	W =  90.000 deg,	P =   0.000 deg,	R =   90.000 deg
};
P[162]{
   GP1:
	UF : 0, UT : 6,		CONFIG : 'N U T, 0, 0, 0',
	X =  224.788  mm,	Y =   -210.243  mm,	Z =   -315.143  mm,
	W =  90.000 deg,	P =   0.000 deg,	R =   90.000 deg
};
P[163]{
   GP1:
	UF : 0, UT : 6,		CONFIG : 'N U T, 0, 0, 0',
	X =  225.758  mm,	Y =   -210.112  mm,	Z =   -326.969  mm,
	W =  90.000 deg,	P =   0.000 deg,	R =   90.000 deg
};
P[164]{
   GP1:
	UF : 0, UT : 6,		CONFIG : 'N U T, 0, 0, 0',
	X =  227.303  mm,	Y =   -209.130  mm,	Z =   -310.855  mm,
	W =  90.000 deg,	P =   0.000 deg,	R =   90.000 deg
};
P[165]{
   GP1:
	UF : 0, UT : 6,		CONFIG : 'N U T, 0, 0, 0',
	X =  228.509  mm,	Y =   -208.538  mm,	Z =   -324.467  mm,
	W =  90.000 deg,	P =   0.000 deg,	R =   90.000 deg
};
P[166]{
   GP1:
	UF : 0, UT : 6,		CONFIG : 'N U T, 0, 0, 0',
	X =  236.027  mm,	Y =   -221.558  mm,	Z =   -327.535  mm,
	W =  90.000 deg,	P =   0.000 deg,	R =   90.000 deg
};
P[167]{
   GP1:
	UF : 0, UT : 6,		CONFIG : 'N U T, 0, 0, 0',
	X =  234.962  mm,	Y =   -222.199  mm,	Z =   -321.974  mm,
	W =  90.000 deg,	P =   0.000 deg,	R =   90.000 deg
};
P[168]{
   GP1:
	UF : 0, UT : 6,		CONFIG : 'N U T, 0, 0, 0',
	X =  234.137  mm,	Y =   -222.880  mm,	Z =   -315.173  mm,
	W =  90.000 deg,	P =   0.000 deg,	R =   90.000 deg
};
P[169]{
   GP1:
	UF : 0, UT : 6,		CONFIG : 'N U T, 0, 0, 0',
	X =  233.285  mm,	Y =   -223.142  mm,	Z =   -324.709  mm,
	W =  90.000 deg,	P =   0.000 deg,	R =   90.000 deg
};
P[170]{
   GP1:
	UF : 0, UT : 6,		CONFIG : 'N U T, 0, 0, 0',
	X =  232.288  mm,	Y =   -223.625  mm,	Z =   -315.398  mm,
	W =  90.000 deg,	P =   0.000 deg,	R =   90.000 deg
};
P[171]{
   GP1:
	UF : 0, UT : 6,		CONFIG : 'N U T, 0, 0, 0',
	X =  231.126  mm,	Y =   -224.281  mm,	Z =   -313.159  mm,
	W =  90.000 deg,	P =   0.000 deg,	R =   90.000 deg
};
P[172]{
   GP1:
	UF : 0, UT : 6,		CONFIG : 'N U T, 0, 0, 0',
	X =  229.645  mm,	Y =   -224.782  mm,	Z =   -313.757  mm,
	W =  90.000 deg,	P =   0.000 deg,	R =   90.000 deg
};
P[173]{
   GP1:
	UF : 0, UT : 6,		CONFIG : 'N U T, 0, 0, 0',
	X =  228.587  mm,	Y =   -225.643  mm,	Z =   -313.551  mm,
	W =  90.000 deg,	P =   0.000 deg,	R =   90.000 deg
};
P[174]{
   GP1:
	UF : 0, UT : 6,		CONFIG : 'N U T, 0, 0, 0',
	X =  228.149  mm,	Y =   -226.124  mm,	Z =   -327.346  mm,
	W =  90.000 deg,	P =   0.000 deg,	R =   90.000 deg
};
P[175]{
   GP1:
	UF : 0, UT : 6,		CONFIG : 'N U T, 0, 0, 0',
	X =  226.254  mm,	Y =   -226.522  mm,	Z =   -322.702  mm,
	W =  90.000 deg,	P =   0.000 deg,	R =   90.000 deg
};
P[176]{
   GP1:
	UF : 0, UT : 6,		CONFIG : 'N U T, 0, 0, 0',
	X =  225.816  mm,	Y =   -227.611  mm,	Z =   -314.588  mm,
	W =  90.000 deg,	P =   0.000 deg,	R =   90.000 deg
};
P[177]{
   GP1:
	UF : 0, UT : 6,		CONFIG : 'N U T, 0, 0, 0',
	X =  224.558  mm,	Y =   -227.894  mm,	Z =   -320.265  mm,
	W =  90.000 deg,	P =   0.000 deg,	R =   90.000 deg
};
P[178]{
   GP1:
	UF : 0, UT : 6,		CONFIG : 'N U T, 0, 0, 0',
	X =  223.276  mm,	Y =   -228.553  mm,	Z =   -326.960  mm,
	W =  90.000 deg,	P =   0.000 deg,	R =   90.000 deg
};
P[179]{
   GP1:
	UF : 0, UT : 6,		CONFIG : 'N U T, 0, 0, 0',
	X =  222.749  mm,	Y =   -229.227  mm,	Z =   -327.686  mm,
	W =  90.000 deg,	P =   0.000 deg,	R =   90.000 deg
};
P[180]{
   GP1:
	UF : 0, UT : 6,		CONFIG : 'N U T, 0, 0, 0',
	X =  221.839  mm,	Y =   -229.266  mm,	Z =   -311.760  mm,
	W =  90.000 deg,	P =   0.000 deg,	R =   90.000 deg
};
P[181]{
   GP1:
	UF : 0, UT : 6,		CONFIG : 'N U T, 0, 0, 0',
	X =  221.094  mm,	Y =   -230.373  mm,	Z =   -313.022  mm,
	W =  90.000 deg,	P =   0.000 deg,	R =   90.000 deg
};
P[182]{
   GP1:
	UF : 0, UT : 6,		CONFIG : 'N U T, 0, 0, 0',
	X =  220.130  mm,	Y =   -230.437  mm,	Z =   -324.917  mm,
	W =  90.000 deg,	P =   0.000 deg,	R =   90.000 deg
};
P[183]{
   GP1:
	UF : 0, UT : 6,		CONFIG : 'N U T, 0, 0, 0',
	X =  219.359  mm,	Y =   -231.525  mm,	Z =   -324.705  mm,
	W =  90.000 deg,	P =   0.000 deg,	R =   90.000 deg
};
P[184]{
   GP1:
	UF : 0, UT : 6,		CONFIG : 'N U T, 0, 0, 0',
	X =  218.328  mm,	Y =   -231.857  mm,	Z =   -320.733  mm,
	W =  90.000 deg,	P =   0.000 deg,	R =   90.000 deg
};
P[185]{
   GP1:
	UF : 0, UT : 6,		CONFIG : 'N U T, 0, 0, 0',
	X =  217.562  mm,	Y =   -231.833  mm,	Z =   -319.447  mm,
	W =  90.000 deg,	P =   0.000 deg,	R =   90.000 deg
};
P[186]{
   GP1:
	UF : 0, UT : 6,		CONFIG : 'N U T, 0, 0, 0',
	X =  216.888  mm,	Y =   -232.430  mm,	Z =   -311.200  mm,
	W =  90.000 deg,	P =   0.000 deg,	R =   90.000 deg
};
P[187]{
   GP1:
	UF : 0, UT : 6,		CONFIG : 'N U T, 0, 0, 0',
	X =  216.001  mm,	Y =   -232.790  mm,	Z =   -327.443  mm,
	W =  90.000 deg,	P =   0.000 deg,	R =   90.000 deg
};
P[188]{
   GP1:
	UF : 0, UT : 6,		CONFIG : 'N U T, 0, 0, 0',
	X =  214.966  mm,	Y =   -233.495  mm,	Z =   -314.364  mm,
	W =  90.000 deg,	P =   0.000 deg,	R =   90.000 deg
};
P[189]{
   GP1:
	UF : 0, UT : 6,		CONFIG : 'N U T, 0, 0, 0',
	X =  213.340  mm,	Y =   -234.714  mm,	Z =   -322.727  mm,
	W =  90.000 deg,	P =   0.000 deg,	R =   90.000 deg
};
P[190]{
   GP1:
	UF : 0, UT : 6,		CONFIG : 'N U T, 0, 0, 0',
	X =  212.316  mm,	Y =   -234.785  mm,	Z =   -314.035  mm,
	W =  90.000 deg,	P =   0.000 deg,	R =   90.000 deg
};
P[191]{
   GP1:
	UF : 0, UT : 6,		CONFIG : 'N U T, 0, 0, 0',
	X =  211.112  mm,	Y =   -235.761  mm,	Z =   -312.348  mm,
	W =  90.000 deg,	P =   0.000 deg,	R =   90.000 deg
};
P[192]{
   GP1:
	UF : 0, UT : 6,		CONFIG : 'N U T, 0, 0, 0',
	X =  209.960  mm,	Y =   -236.382  mm,	Z =   -315.125  mm,
	W =  90.000 deg,	P =   0.000 deg,	R =   90.000 deg
};
P[193]{
   GP1:
	UF : 0, UT : 6,		CONFIG : 'N U T, 0, 0, 0',
	X =  209.037  mm,	Y =   -237.118  mm,	Z =   -320.198  mm,
	W =  90.000 deg,	P =   0.000 deg,	R =   90.000 deg
};
P[194]{
   GP1:
	UF : 0, UT : 6,		CONFIG : 'N U T, 0, 0, 0',
	X =  208.026  mm,	Y =   -237.481  mm,	Z =   -316.356  mm,
	W =  90.000 deg,	P =   0.000 deg,	R =   90.000 deg
};
P[195]{
   GP1:
	UF : 0, UT : 6,		CONFIG : 'N U T, 0, 0, 0',
	X =  207.935  mm,	Y =   -238.178  mm,	Z =   -325.493  mm,
	W =  90.000 deg,	P =   0.000 deg,	R =   90.000 deg
};
P[196]{
   GP1:
	UF : 0, UT : 6,		CONFIG : 'N U T, 0, 0, 0',
	X =  207.107  mm,	Y =   -237.985  mm,	Z =   -319.169  mm,
	W =  90.000 deg,	P =   0.000 deg,	R =   90.000 deg
};
P[197]{
   GP1:
	UF : 0, UT : 6,		CONFIG : 'N U T, 0, 0, 0',
	X =  207.148  mm,	Y =   -238.292  mm,	Z =   -322.311  mm,
	W =  90.000 deg,	P =   0.000 deg,	R =   90.000 deg
};
P[198]{
   GP1:
	UF : 0, UT : 6,		CONFIG : 'N U T, 0, 0, 0',
	X =  207.193  mm,	Y =   -238.442  mm,	Z =   -317.365  mm,
	W =  90.000 deg,	P =   0.000 deg,	R =   90.000 deg
};
P[199]{
   GP1:
	UF : 0, UT : 6,		CONFIG : 'N U T, 0, 0, 0',
	X =  207.015  mm,	Y =   -238.202  mm,	Z =   -313.956  mm,
	W =  90.000 deg,	P =   0.000 deg,	R =   90.000 deg
};
P[200]{
   GP1:
	UF : 0, UT : 6,		CONFIG : 'N U T, 0, 0, 0',
	X =  206.545  mm,	Y =   -238.830  mm,	Z =   -313.041  mm,
	W =  90.000 deg,	P =   0.000 deg,	R =   90.000 deg
};
P[201]{
   GP1:
	UF : 0, UT : 6,		CONFIG : 'N U T, 0, 0, 0',
	X =  206.046  mm,	Y =   -238.312  mm,	Z =   -321.821  mm,
	W =  90.000 deg,	P =   0.000 deg,	R =   90.000 deg
};
P[202]{
   GP1:
	UF : 0, UT : 6,		CONFIG : 'N U T, 0, 0, 0',
	X =  206.072  mm,	Y =   -238.413  mm,	Z =   -313.566  mm,
	W =  90.000 deg,	P =   0.000 deg,	R =   90.000 deg
};
P[203]{
   GP1:
	UF : 0, UT : 6,		CONFIG : 'N U T, 0, 0, 0',
	X =  206.000  mm,	Y =   -238.618  mm,	Z =   -319.197  mm,
	W =  90.000 deg,	P =   0.000 deg,	R =   90.000 deg
};
P[204]{
   GP1:
	UF : 0, UT : 6,		CONFIG : 'N U T, 0, 0, 0',
	X =  205.360  mm,	Y =   -238.553  mm,	Z =   -323.476  mm,
	W =  90.000 deg,	P =   0.000 deg,	R =   90.000 deg
};
P[205]{
   GP1:
	UF : 0, UT : 6,		CONFIG : 'N U T, 0, 0, 0',
	X =  205.394  mm,	Y =   -238.816  mm,	Z =   -314.327  mm,
	W =  90.000 deg,	P =   0.000 deg,	R =   90.000 deg
};
P[206]{
   GP1:
	UF : 0, UT : 6,		CONFIG : 'N U T, 0, 0, 0',
	X =  205.468  mm,	Y =   -239.148  mm,	Z =   -318.562  mm,
	W =  90.000 deg,	P =   0.000 deg,	R =   90.000 deg
};
P[207]{
   GP1:
	UF : 0, UT : 6,		CONFIG : 'N U T, 0, 0, 0',
	X =  205.209  mm,	Y =   -239.739  mm,	Z =   -324.188  mm,
	W =  90.000 deg,	P =   0.000 deg,	R =   90.000 deg
};
P[208]{
   GP1:
	UF : 0, UT : 6,		CONFIG : 'N U T, 0, 0, 0',
	X =  204.658  mm,	Y =   -239.589  mm,	Z =   -316.726  mm,
	W =  90.000 deg,	P =   0.000 deg,	R =   90.000 deg
};
P[209]{
   GP1:
	UF : 0, UT : 6,		CONFIG : 'N U T, 0, 0, 0',
	X =  203.848  mm,	Y =   -239.576  mm,	Z =   -324.082  mm,
	W =  90.000 deg,	P =   0.000 deg,	R =   90.000 deg
};
P[210]{
   GP1:
	UF : 0, UT : 6,		CONFIG : 'N U T, 0, 0, 0',
	X =  203.724  mm,	Y =   -240.092  mm,	Z =   -313.323  mm,
	W =  90.000 deg,	P =   0.000 deg,	R =   90.000 deg
};
P[211]{
   GP1:
	UF : 0, UT : 6,		CONFIG : 'N U T, 0, 0, 0',
	X =  202.753  mm,	Y =   -240.091  mm,	Z =   -323.496  mm,
	W =  90.000 deg,	P =   0.000 deg,	R =   90.000 deg
};
P[212]{
   GP1:
	UF : 0, UT : 6,		CONFIG : 'N U T, 0, 0, 0',
	X =  202.841  mm,	Y =   -240.719  mm,	Z =   -325.615  mm,
	W =  90.000 deg,	P =   0.000 deg,	R =   90.000 deg
};
P[213]{
   GP1:
	UF : 0, UT : 6,		CONFIG : 'N U T, 0, 0, 0',
	X =  202.714  mm,	Y =   -241.173  mm,	Z =   -323.812  mm,
	W =  90.000 deg,	P =   0.000 deg,	R =   90.000 deg
};
P[214]{
   GP1:
	UF : 0, UT : 6,		CONFIG : 'N U T, 0, 0, 0',
	X =  202.146  mm,	Y =   -240.408  mm,	Z =   -321.973  mm,
	W =  90.000 deg,	P =   0.000 deg,	R =   90.000 deg
};
P[215]{
   GP1:
	UF : 0, UT : 6,		CONFIG : 'N U T, 0, 0, 0',
	X =  202.040  mm,	Y =   -241.144  mm,	Z =   -319.450  mm,
	W =  90.000 deg,	P =   0.000 deg,	R =   90.000 deg
};
P[216]{
   GP1:
	UF : 0, UT : 6,		CONFIG : 'N U T, 0, 0, 0',
	X =  201.603  mm,	Y =   -240.788  mm,	Z =   -326.320  mm,
	W =  90.000 deg,	P =   0.000 deg,	R =   90.000 deg
};
P[217]{
   GP1:
	UF : 0, UT : 6,		CONFIG : 'N U T, 0, 0, 0',
	X =  200.943  mm,	Y =   -241.147  mm,	Z =   -325.486  mm,
	W =  90.000 deg,	P =   0.000 deg,	R =   90.000 deg
};
P[218]{
   GP1:
	UF : 0, UT : 6,		CONFIG : 'N U T, 0, 0, 0',
	X =  201.039  mm,	Y =   -241.818  mm,	Z =   -323.445  mm,
	W =  90.000 deg,	P =   0.000 deg,	R =   90.000 deg
};
P[219]{
   GP1:
	UF : 0, UT : 6,		CONFIG : 'N U T, 0, 0, 0',
	X =  200.525  mm,	Y =   -241.662  mm,	Z =   -318.426  mm,
	W =  90.000 deg,	P =   0.000 deg,	R =   90.000 deg
};
P[220]{
   GP1:
	UF : 0, UT : 6,		CONFIG : 'N U T, 0, 0, 0',
	X =  200.346  mm,	Y =   -242.443  mm,	Z =   -322.944  mm,
	W =  90.000 deg,	P =   0.000 deg,	R =   90.000 deg
};
P[221]{
   GP1:
	UF : 0, UT : 6,		CONFIG : 'N U T, 0, 0, 0',
	X =  199.677  mm,	Y =   -242.289  mm,	Z =   -319.034  mm,
	W =  90.000 deg,	P =   0.000 deg,	R =   90.000 deg
};
P[222]{
   GP1:
	UF : 0, UT : 6,		CONFIG : 'N U T, 0, 0, 0',
	X =  198.880  mm,	Y =   -243.196  mm,	Z =   -312.137  mm,
	W =  90.000 deg,	P =   0.000 deg,	R =   90.000 deg
};
P[223]{
   GP1:
	UF : 0, UT : 6,		CONFIG : 'N U T, 0, 0, 0',
	X =  198.372  mm,	Y =   -242.908  mm,	Z =   -319.670  mm,
	W =  90.000 deg,	P =   0.000 deg,	R =   90.000 deg
};
P[224]{
   GP1:
	UF : 0, UT : 6,		CONFIG : 'N U T, 0, 0, 0',
	X =  197.548  mm,	Y =   -243.227  mm,	Z =   -320.526  mm,
	W =  90.000 deg,	P =   0.000 deg,	R =   90.000 deg
};
P[225]{
   GP1:
	UF : 0, UT : 6,		CONFIG : 'N U T, 0, 0, 0',
	X =  197.608  mm,	Y =   -243.970  mm,	Z =   -310.144  mm,
	W =  90.000 deg,	P =   0.000 deg,	R =   90.000 deg
};
P[226]{
   GP1:
	UF : 0, UT : 6,		CONFIG : 'N U T, 0, 0, 0',
	X =  196.892  mm,	Y =   -244.207  mm,	Z =   -322.889  mm,
	W =  90.000 deg,	P =   0.000 deg,	R =   90.000 deg
};
P[227]{
   GP1:
	UF : 0, UT : 6,		CONFIG : 'N U T, 0, 0, 0',
	X =  195.770  mm,	Y =   -244.534  mm,	Z =   -317.358  mm,
	W =  90.000 deg,	P =   0.000 deg,	R =   90.000 deg
};
P[228]{
   GP1:
	UF : 0, UT : 6,		CONFIG : 'N U T, 0, 0, 0',
	X =  195.153  mm,	Y =   -245.287  mm,	Z =   -316.689  mm,
	W =  90.000 deg,	P =   0.000 deg,	R =   90.000 deg
};
P[229]{
   GP1:
	UF : 0, UT : 6,		CONFIG : 'N U T, 0, 0, 0',
	X =  194.505  mm,	Y =   -244.820  mm,	Z =   -323.698  mm,
	W =  90.000 deg,	P =   0.000 deg,	R =   90.000 deg
};
P[230]{
   GP1:
	UF : 0, UT : 6,		CONFIG : 'N U T, 0, 0, 0',
	X =  194.224  mm,	Y =   -245.716  mm,	Z =   -326.476  mm,
	W =  90.000 deg,	P =   0.000 deg,	R =   90.000 deg
};
P[231]{
   GP1:
	UF : 0, UT : 6,		CONFIG : 'N U T, 0, 0, 0',
	X =  193.462  mm,	Y =   -245.718  mm,	Z =   -315.944  mm,
	W =  90.000 deg,	P =   0.000 deg,	R =   90.000 deg
};
P[232]{
   GP1:
	UF : 0, UT : 6,		CONFIG : 'N U T, 0, 0, 0',
	X =  193.608  mm,	Y =   -246.149  mm,	Z =   -317.665  mm,
	W =  90.000 deg,	P =   0.000 deg,	R =   90.000 deg
};
P[233]{
   GP1:
	UF : 0, UT : 6,		CONFIG : 'N U T, 0, 0, 0',
	X =  192.403  mm,	Y =   -246.571  mm,	Z =   -321.320  mm,
	W =  90.000 deg,	P =   0.000 deg,	R =   90.000 deg
};
P[234]{
   GP1:
	UF : 0, UT : 6,		CONFIG : 'N U T, 0, 0, 0',
	X =  191.248  mm,	Y =   -247.020  mm,	Z =   -319.008  mm,
	W =  90.000 deg,	P =   0.000 deg,	R =   90.000 deg
};
P[235]{
   GP1:
	UF : 0, UT : 6,		CONFIG : 'N U T, 0, 0, 0',
	X =  191.043  mm,	Y =   -247.641  mm,	Z =   -317.853  mm,
	W =  90.000 deg,	P =   0.000 deg,	R =   90.000 deg
};
P[236]{
   GP1:
	UF : 0, UT : 6,		CONFIG : 'N U T, 0, 0, 0',
	X =  190.516  mm,	Y =   -247.406  mm,	Z =   -314.457  mm,
	W =  90.000 deg,	P =   0.000 deg,	R =   90.000 deg
};
P[237]{
   GP1:
	UF : 0, UT : 6,		CONFIG : 'N U T, 0, 0, 0',
	X =  189.836  mm,	Y =   -248.145  mm,	Z =   -315.818  mm,
	W =  90.000 deg,	P =   0.000 deg,	R =   90.000 deg
};
P[238]{
   GP1:
	UF : 0, UT : 6,		CONFIG : 'N U T, 0, 0, 0',
	X =  189.085  mm,	Y =   -248.519  mm,	Z =   -310.157  mm,
	W =  90.000 deg,	P =   0.000 deg,	R =   90.000 deg
};
P[239]{
   GP1:
	UF : 0, UT : 6,		CONFIG : 'N U T, 0, 0, 0',
	X =  188.507  mm,	Y =   -248.566  mm,	Z =   -315.070  mm,
	W =  90.000 deg,	P =   0.000 deg,	R =   90.000 deg
};
P[240]{
   GP1:
	UF : 0, UT : 6,		CONFIG : 'N U T, 0, 0, 0',
	X =  187.787  mm,	Y =   -248.752  mm,	Z =   -325.940  mm,
	W =  90.000 deg,	P =   0.000 deg,	R =   90.000 deg
};
P[241]{
   GP1:
	UF : 0, UT : 6,		CONFIG : 'N U T, 0, 0, 0',
	X =  187.122  mm,	Y =   -249.652  mm,	Z =   -310.999  mm,
	W =  90.000 deg,	P =   0.000 deg,	R =   90.000 deg
};
P[242]{
   GP1:
	UF : 0, UT : 6,		CONFIG : 'N U T, 0, 0, 0',
	X =  186.808  mm,	Y =   -250.365  mm,	Z =   -322.828  mm,
	W =  90.000 deg,	P =   0.000 deg,	R =   90.000 deg
};
P[243]{
   GP1:
	UF : 0, UT : 6,		CONFIG : 'N U T, 0, 0, 0',
	X =  186.334  mm,	Y =   -249.614  mm,	Z =   -326.737  mm,
	W =  90.000 deg,	P =   0.000 deg,	R =   90.000 deg
};
P[244]{
   GP1:
	UF : 0, UT : 6,		CONFIG : 'N U T, 0, 0, 0',
	X =  186.496  mm,	Y =   -249.995  mm,	Z =   -310.681  mm,
	W =  90.000 deg,	P =   0.000 deg,	R =   90.000 deg
};
P[245]{
   GP1:
	UF : 0, UT : 6,		CONFIG : 'N U T, 0, 0, 0',
	X =  185.651  mm,	Y =   -250.675  mm,	Z =   -324.252  mm,
	W =  90.000 deg,	P =   0.000 deg,	R =   90.000 deg
};
P[246]{
   GP1:
	UF : 0, UT : 6,		CONFIG : 'N U T, 0, 0, 0',
	X =  185.181  mm,	Y =   -250.524  mm,	Z =   -319.591  mm,
	W =  90.000 deg,	P =   0.000 deg,	R =   90.000 deg
};
P[247]{
   GP1:
	UF : 0, UT : 6,		CONFIG : 'N U T, 0, 0, 0',
	X =  184.766  mm,	Y =   -251.330  mm,	Z =   -314.019  mm,
	W =  90.000 deg,	P =   0.000 deg,	R =   90.000 deg
};
P[248]{
   GP1:
	UF : 0, UT : 6,		CONFIG : 'N U T, 0, 0, 0',
	X =  184.217  mm,	Y =   -251.057  mm,	Z =   -315.680  mm,
	W =  90.000 deg,	P =   0.000 deg,	R =   90.000 deg
};
P[249]{
   GP1:
	UF : 0, UT : 6,		CONFIG : 'N U T, 0, 0, 0',
	X =  183.503  mm,	Y =   -251.481  mm,	Z =   -319.071  mm,
	W =  90.000 deg,	P =   0.000 deg,	R =   90.000 deg
};
P[250]{
   GP1:
	UF : 0, UT : 6,		CONFIG : 'N U T, 0, 0, 0',
	X =  183.596  mm,	Y =   -252.173  mm,	Z =   -323.935  mm,
	W =  90.000 deg,	P =   0.000 deg,	R =   90.000 deg
};
P[251]{
   GP1:
	UF : 0, UT : 6,		CONFIG : 'N U T, 0, 0, 0',
	X =  182.808  mm,	Y =   -251.854  mm,	Z =   -313.115  mm,
	W =  90.000 deg,	P =   0.000 deg,	R =   90.000 deg
};
P[252]{
   GP1:
	UF : 0, UT : 6,		CONFIG : 'N U T, 0, 0, 0',
	X =  182.519  mm,	Y =   -252.698  mm,	Z =   -311.094  mm,
	W =  90.000 deg,	P =   0.000 deg,	R =   90.000 deg
};
P[253]{
   GP1:
	UF : 0, UT : 6,		CONFIG : 'N U T, 0, 0, 0',
	X =  182.133  mm,	Y =   -252.554  mm,	Z =   -312.961  mm,
	W =  90.000 deg,	P =   0.000 deg,	R =   90.000 deg
};
P[254]{
   GP1:
	UF : 0, UT : 6,		CONFIG : 'N U T, 0, 0, 0',
	X =  181.696  mm,	Y =   -252.481  mm,	Z =   -312.907  mm,
	W =  90.000 deg,	P =   0.000 deg,	R =   90.000 deg
};
P[255]{
   GP1:
	UF : 0, UT : 6,		CONFIG : 'N U T, 0, 0, 0',
	X =  181.475  mm,	Y =   -253.156  mm,	Z =   -318.417  mm,
	W =  90.000 deg,	P =   0.000 deg,	R =   90.000 deg
};
P[256]{
   GP1:
	UF : 0, UT : 6,		CONFIG : 'N U T, 0, 0, 0',
	X =  181.098  mm,	Y =   -252.670  mm,	Z =   -325.683  mm,
	W =  90.000 deg,	P =   0.000 deg,	R =   90.000 deg
};
P[257]{
   GP1:
	UF : 0, UT : 6,		CONFIG : 'N U T, 0, 0, 0',
	X =  180.715  mm,	Y =   -253.461  mm,	Z =   -319.202  mm,
	W =  90.000 deg,	P =   0.000 deg,	R =   90.000 deg
};
P[258]{
   GP1:
	UF : 0, UT : 6,		CONFIG : 'N U T, 0, 0, 0',
	X =  180.117  mm,	Y =   -253.445  mm,	Z =   -316.961  mm,
	W =  90.000 deg,	P =   0.000 deg,	R =   90.000 deg
};
P[259]{
   GP1:
	UF : 0, UT : 6,		CONFIG : 'N U T, 0, 0, 0',
	X =  179.724  mm,	Y =   -253.405  mm,	Z =   -327.050  mm,
	W =  90.000 deg,	P =   0.000 deg,	R =   90.000 deg
};
P[260]{
   GP1:
	UF : 0, UT : 6,		CONFIG : 'N U T, 0, 0, 0',
	X =  179.758  mm,	Y =   -254.263  mm,	Z =   -310.411  mm,
	W =  90.000 deg,	P =   0.000 deg,	R =   90.000 deg
};
P[261]{
   GP1:
	UF : 0, UT : 6,		CONFIG : 'N U T, 0, 0, 0',
	X =  179.421  mm,	Y =   -254.004  mm,	Z =   -316.422  mm,
	W =  90.000 deg,	P =   0.000 deg,	R =   90.000 deg
};
P[262]{
   GP1:
	UF : 0, UT : 6,		CONFIG : 'N U T, 0, 0, 0',
	X =  179.168  mm,	Y =   -254.767  mm,	Z =   -323.170  mm,
	W =  90.000 deg,	P =   0.000 deg,	R =   90.000 deg
};
P[263]{
   GP1:
	UF : 0, UT : 6,		CONFIG : 'N U T, 0, 0, 0',
	X =  178.774  mm,	Y =   -254.695  mm,	Z =   -320.156  mm,
	W =  90.000 deg,	P =   0.000 deg,	R =   90.000 deg
};
P[264]{
   GP1:
	UF : 0, UT : 6,		CONFIG : 'N U T, 0, 0, 0',
	X =  178.329  mm,	Y =   -254.157  mm,	Z =   -322.081  mm,
	W =  90.000 deg,	P =   0.000 deg,	R =   90.000 deg
};
P[265]{
   GP1:
	UF : 0, UT : 6,		CONFIG : 'N U T, 0, 0, 0',
	X =  178.522  mm,	Y =   -254.533  mm,	Z =   -316.123  mm,
	W =  90.000 deg,	P =   0.000 deg,	R =   90.000 deg
};
P[266]{
   GP1:
	UF : 0, UT : 6,		CONFIG : 'N U T, 0, 0, 0',
	X =  177.645  mm,	Y =   -254.955  mm,	Z =   -324.671  mm,
	W =  90.000 deg,	P =   0.000 deg,	R =   90.000 deg
};
P[267]{
   GP1:
	UF : 0, UT : 6,		CONFIG : 'N U T, 0, 0, 0',
	X =  177.564  mm,	Y =   -255.635  mm,	Z =   -326.048  mm,
	W =  90.000 deg,	P =   0.000 deg,	R =   90.000 deg
};
P[268]{
   GP1:
	UF : 0, UT : 6,		CONFIG : 'N U T, 0, 0, 0',
	X =  176.916  mm,	Y =   -255.259  mm,	Z =   -314.337  mm,
	W =  90.000 deg,	P =   0.000 deg,	R =   90.000 deg
};
P[269]{
   GP1:
	UF : 0, UT : 6,		CONFIG : 'N U T, 0, 0, 0',
	X =  176.707  mm,	Y =   -256.020  mm,	Z =   -311.027  mm,
	W =  90.000 deg,	P =   0.000 deg,	R =   90.000 deg
};
P[270]{
   GP1:
	UF : 0, UT : 6,		CONFIG : 'N U T, 0, 0, 0',
	X =  176.355  mm,	Y =   -255.557  mm,	Z =   -312.955  mm,
	W =  90.000 deg,	P =   0.000 deg,	R =   90.000 deg
};
P[271]{
   GP1:
	UF : 0, UT : 6,		CONFIG : 'N U T, 0, 0, 0',
	X =  176.055  mm,	Y =   -256.024  mm,	Z =   -309.916  mm,
	W =  90.000 deg,	P =   0.000 deg,	R =   90.000 deg
};
P[272]{
   GP1:
	UF : 0, UT : 6,		CONFIG : 'N U T, 0, 0, 0',
	X =  176.130  mm,	Y =   -256.296  mm,	Z =   -315.346  mm,
	W =  90.000 deg,	P =   0.000 deg,	R =   90.000 deg
};
P[273]{
   GP1:
	UF : 0, UT : 6,		CONFIG : 'N U T, 0, 0, 0',
	X =  175.786  mm,	Y =   -255.774  mm,	Z =   -322.730  mm,
	W =  90.000 deg,	P =   0.000 deg,	R =   90.000 deg
};
P[274]{
   GP1:
	UF : 0, UT : 6,		CONFIG : 'N U T, 0, 0, 0',
	X =  175.133  mm,	Y =   -256.020  mm,	Z =   -323.009  mm,
	W =  90.000 deg,	P =   0.000 deg,	R =   90.000 deg
};
P[275]{
   GP1:
	UF : 0, UT : 6,		CONFIG : 'N U T, 0, 0, 0',
	X =  175.034  mm,	Y =   -256.520  mm,	Z =   -318.149  mm,
	W =  90.000 deg,	P =   0.000 deg,	R =   90.000 deg
};
P[276]{
   GP1:
	UF : 0, UT : 6,		CONFIG : 'N U T, 0, 0, 0',
	X =  174.768  mm,	Y =   -256.256  mm,	Z =   -327.394  mm,
	W =  90.000 deg,	P =   0.000 deg,	R =   90.000 deg
};
P[277]{
   GP1:
	UF : 0, UT : 6,		CONFIG : 'N U T, 0, 0, 0',
	X =  175.139  mm,	Y =   -257.050  mm,	Z =   -326.450  mm,
	W =  90.000 deg,	P =   0.000 deg,	R =   90.000 deg
};
P[278]{
   GP1:
	UF : 0, UT : 6,		CONFIG : 'N U T, 0, 0, 0',
	X =  174.185  mm,	Y =   -257.011  mm,	Z =   -318.021  mm,
	W =  90.000 deg,	P =   0.000 deg,	R =   90.000 deg
};
P[279]{
   GP1:
	UF : 0, UT : 6,		CONFIG : 'N U T, 0, 0, 0',
	X =  174.073  mm,	Y =   -256.837  mm,	Z =   -310.875  mm,
	W =  90.000 deg,	P =   0.000 deg,	R =   90.000 deg
};
P[280]{
   GP1:
	UF : 0, UT : 6,		CONFIG : 'N U T, 0, 0, 0',
	X =  173.977  mm,	Y =   -256.815  mm,	Z =   -323.368  mm,
	W =  90.000 deg,	P =   0.000 deg,	R =   90.000 deg
};
P[281]{
   GP1:
	UF : 0, UT : 6,		CONFIG : 'N U T, 0, 0, 0',
	X =  174.328  mm,	Y =   -257.478  mm,	Z =   -322.177  mm,
	W =  90.000 deg,	P =   0.000 deg,	R =   90.000 deg
};
P[282]{
   GP1:
	UF : 0, UT : 6,		CONFIG : 'N U T, 0, 0, 0',
	X =  173.792  mm,	Y =   -256.836  mm,	Z =   -326.792  mm,
	W =  90.000 deg,	P =   0.000 deg,	R =   90.000 deg
};
P[283]{
   GP1:
	UF : 0, UT : 6,		CONFIG : 'N U T, 0, 0, 0',
	X =  174.088  mm,	Y =   -257.395  mm,	Z =   -320.324  mm,
	W =  90.000 deg,	P =   0.000 deg,	R =   90.000 deg
};
P[284]{
   GP1:
	UF : 0, UT : 6,		CONFIG : 'N U T, 0, 0, 0',
	X =  173.281  mm,	Y =   -257.367  mm,	Z =   -315.190  mm,
	W =  90.000 deg,	P =   0.000 deg,	R =   90.000 deg
};
P[285]{
   GP1:
	UF : 0, UT : 6,		CONFIG : 'N U T, 0, 0, 0',
	X =  173.246  mm,	Y =   -257.556  mm,	Z =   -317.174  mm,
	W =  90.000 deg,	P =   0.000 deg,	R =   90.000 deg
};
P[286]{
   GP1:
	UF : 0, UT : 6,		CONFIG : 'N U T, 0, 0, 0',
	X =  173.451  mm,	Y =   -258.059  mm,	Z =   -323.350  mm,
	W =  90.000 deg,	P =   0.000 deg,	R =   90.000 deg
};
P[287]{
   GP1:
	UF : 0, UT : 6,		CONFIG : 'N U T, 0, 0, 0',
	X =  172.991  mm,	Y =   -257.452  mm,	Z =   -311.441  mm,
	W =  90.000 deg,	P =   0.000 deg,	R =   90.000 deg
};
P[288]{
   GP1:
	UF : 0, UT : 6,		CONFIG : 'N U T, 0, 0, 0',
	X =  172.967  mm,	Y =   -257.956  mm,	Z =   -327.172  mm,
	W =  90.000 deg,	P =   0.000 deg,	R =   90.000 deg
};
P[289]{
   GP1:
	UF : 0, UT : 6,		CONFIG : 'N U T, 0, 0, 0',
	X =  172.399  mm,	Y =   -258.123  mm,	Z =   -325.331  mm,
	W =  90.000 deg,	P =   0.000 deg,	R =   90.000 deg
};
P[290]{
   GP1:
	UF : 0, UT : 6,		CONFIG : 'N U T, 0, 0, 0',
	X =  172.171  mm,	Y =   -258.662  mm,	Z =   -320.276  mm,
	W =  90.000 deg,	P =   0.000 deg,	R =   90.000 deg
};
P[291]{
   GP1:
	UF : 0, UT : 6,		CONFIG : 'N U T, 0, 0, 0',
	X =  171.769  mm,	Y =   -258.821  mm,	Z =   -313.988  mm,
	W =  90.000 deg,	P =   0.000 deg,	R =   90.000 deg
};
P[292]{
   GP1:
	UF : 0, UT : 6,		CONFIG : 'N U T, 0, 0, 0',
	X =  171.718  mm,	Y =   -258.746  mm,	Z =   -323.267  mm,
	W =  90.000 deg,	P =   0.000 deg,	R =   90.000 deg
};
P[293]{
   GP1:
	UF : 0, UT : 6,		CONFIG : 'N U T, 0, 0, 0',
	X =  171.315  mm,	Y =   -258.833  mm,	Z =   -316.420  mm,
	W =  90.000 deg,	P =   0.000 deg,	R =   90.000 deg
};
P[294]{
   GP1:
	UF : 0, UT : 6,		CONFIG : 'N U T, 0, 0, 0',
	X =  171.438  mm,	Y =   -259.276  mm,	Z =   -321.449  mm,
	W =  90.000 deg,	P =   0.000 deg,	R =   90.000 deg
};
P[295]{
   GP1:
	UF : 0, UT : 6,		CONFIG : 'N U T, 0, 0, 0',
	X =  170.919  mm,	Y =   -259.359  mm,	Z =   -310.652  mm,
	W =  90.000 deg,	P =   0.000 deg,	R =   90.000 deg
};
P[296]{
   GP1:
	UF : 0, UT : 6,		CONFIG : 'N U T, 0, 0, 0',
	X =  170.435  mm,	Y =   -258.753  mm,	Z =   -323.064  mm,
	W =  90.000 deg,	P =   0.000 deg,	R =   90.000 deg
};
P[297]{
   GP1:
	UF : 0, UT : 6,		CONFIG : 'N U T, 0, 0, 0',
	X =  170.812  mm,	Y =   -259.537  mm,	Z =   -326.812  mm,
	W =  90.000 deg,	P =   0.000 deg,	R =   90.000 deg
};
P[298]{
   GP1:
	UF : 0, UT : 6,		CONFIG : 'N U T, 0, 0, 0',
	X =  170.323  mm,	Y =   -259.748  mm,	Z =   -322.919  mm,
	W =  90.000 deg,	P =   0.000 deg,	R =   90.000 deg
};
P[299]{
   GP1:
	UF : 0, UT : 6,		CONFIG : 'N U T, 0, 0, 0',
	X =  169.161  mm,	Y =   -260.175  mm,	Z =   -326.899  mm,
	W =  90.000 deg,	P =   0.000 deg,	R =   90.000 deg
};
P[300]{
   GP1:
	UF : 0, UT : 6,		CONFIG : 'N U T, 0, 0, 0',
	X =  168.079  mm,	Y =   -260.866  mm,	Z =   -320.051  mm,
	W =  90.000 deg,	P =   0.000 deg,	R =   90.000 deg
};
P[301]{
   GP1:
	UF : 0, UT : 6,		CONFIG : 'N U T, 0, 0, 0',
	X =  167.000  mm,	Y =   -261.260  mm,	Z =   -310.192  mm,
	W =  90.000 deg,	P =   0.000 deg,	R =   90.000 deg
};
P[302]{
   GP1:
	UF : 0, UT : 6,		CONFIG : 'N U T, 0, 0, 0',
	X =  165.759  mm,	Y =   -261.835  mm,	Z =   -322.908  mm,
	W =  90.000 deg,	P =   0.000 deg,	R =   90.000 deg
};
P[303]{
   GP1:
	UF : 0, UT : 6,		CONFIG : 'N U T, 0, 0, 0',
	X =  164.606  mm,	Y =   -262.570  mm,	Z =   -315.081  mm,
	W =  90.000 deg,	P =   0.000 deg,	R =   90.000 deg
};
P[304]{
   GP1:
	UF : 0, UT : 6,		CONFIG : 'N U T, 0, 0, 0',
	X =  163.888  mm,	Y =   -263.372  mm,	Z =   -314.268  mm,
	W =  90.000 deg,	P =   0.000 deg,	R =   90.000 deg
};
P[305]{
   GP1:
	UF : 0, UT : 6,		CONFIG : 'N U T, 0, 0, 0',
	X =  163.182  mm,	Y =   -263.663  mm,	Z =   -322.510  mm,
	W =  90.000 deg,	P =   0.000 deg,	R =   90.000 deg
};
P[306]{
   GP1:
	UF : 0, UT : 6,		CONFIG : 'N U T, 0, 0, 0',
	X =  162.268  mm,	Y =   -264.286  mm,	Z =   -315.824  mm,
	W =  90.000 deg,	P =   0.000 deg,	R =   90.000 deg
};
P[307]{
   GP1:
	UF : 0, UT : 6,		CONFIG : 'N U T, 0, 0, 0',
	X =  161.046  mm,	Y =   -264.171  mm,	Z =   -324.463  mm,
	W =  90.000 deg,	P =   0.000 deg,	R =   90.000 deg
};
P[308]{
   GP1:
	UF : 0, UT : 6,		CONFIG : 'N U T, 0, 0, 0',
	X =  160.503  mm,	Y =   -264.987  mm,	Z =   -310.228  mm,
	W =  90.000 deg,	P =   0.000 deg,	R =   90.000 deg
};
P[309]{
   GP1:
	UF : 0, UT : 6,		CONFIG : 'N U T, 0, 0, 0',
	X =  159.727  mm,	Y =   -265.455  mm,	Z =   -311.043  mm,
	W =  90.000 deg,	P =   0.000 deg,	R =   90.000 deg
};
P[310]{
   GP1:
	UF : 0, UT : 6,		CONFIG : 'N U T, 0, 0, 0',
	X =  158.548  mm,	Y =   -265.744  mm,	Z =   -324.807  mm,
	W =  90.000 deg,	P =   0.000 deg,	R =   90.000 deg
};
P[311]{
   GP1:
	UF : 0, UT : 6,		CONFIG : 'N U T, 0, 0, 0',
	X =  157.941  mm,	Y =   -266.872  mm,	Z =   -309.962  mm,
	W =  90.000 deg,	P =   0.000 deg,	R =   90.000 deg
};
P[312]{
   GP1:
	UF : 0, UT : 6,		CONFIG : 'N U T, 0, 0, 0',
	X =  155.789  mm,	Y =   -267.639  mm,	Z =   -316.630  mm,
	W =  90.000 deg,	P =   0.000 deg,	R =   90.000 deg
};
P[313]{
   GP1:
	UF : 0, UT : 6,		CONFIG : 'N U T, 0, 0, 0',
	X =  155.104  mm,	Y =   -268.015  mm,	Z =   -318.141  mm,
	W =  90.000 deg,	P =   0.000 deg,	R =   90.000 deg
};
P[314]{
   GP1:
	UF : 0, UT : 6,		CONFIG : 'N U T, 0, 0, 0',
	X =  154.627  mm,	Y =   -268.796  mm,	Z =   -316.149  mm,
	W =  90.000 deg,	P =   0.000 deg,	R =   90.000 deg
};
P[315]{
   GP1:
	UF : 0, UT : 6,		CONFIG : 'N U T, 0, 0, 0',
	X =  152.644  mm,	Y =   -269.405  mm,	Z =   -325.490  mm,
	W =  90.000 deg,	P =   0.000 deg,	R =   90.000 deg
};
P[316]{
   GP1:
	UF : 0, UT : 6,		CONFIG : 'N U T, 0, 0, 0',
	X =  151.708  mm,	Y =   -270.168  mm,	Z =   -316.163  mm,
	W =  90.000 deg,	P =   0.000 deg,	R =   90.000 deg
};
P[317]{
   GP1:
	UF : 0, UT : 6,		CONFIG : 'N U T, 0, 0, 0',
	X =  151.058  mm,	Y =   -270.792  mm,	Z =   -313.563  mm,
	W =  90.000 deg,	P =   0.000 deg,	R =   90.000 deg
};
P[318]{
   GP1:
	UF : 0, UT : 6,		CONFIG : 'N U T, 0, 0, 0',
	X =  150.279  mm,	Y =   -270.993  mm,	Z =   -316.136  mm,
	W =  90.000 deg,	P =   0.000 deg,	R =   90.000 deg
};
P[319]{
   GP1:
	UF : 0, UT : 6,		CONFIG : 'N U T, 0, 0, 0',
	X =  148.923  mm,	Y =   -271.261  mm,	Z =   -321.051  mm,
	W =  90.000 deg,	P =   0.000 deg,	R =   90.000 deg
};
P[320]{
   GP1:
	UF : 0, UT : 6,		CONFIG : 'N U T, 0, 0, 0',
	X =  148.393  mm,	Y =   -272.295  mm,	Z =   -315.157  mm,
	W =  90.000 deg,	P =   0.000 deg,	R =   90.000 deg
};
P[321]{
   GP1:
	UF : 0, UT : 6,		CONFIG : 'N U T, 0, 0, 0',
	X =  147.670  mm,	Y =   -272.189  mm,	Z =   -320.863  mm,
	W =  90.000 deg,	P =   0.000 deg,	R =   90.000 deg
};
P[322]{
   GP1:
	UF : 0, UT : 6,		CONFIG : 'N U T, 0, 0, 0',
	X =  146.965  mm,	Y =   -273.156  mm,	Z =   -314.071  mm,
	W =  90.000 deg,	P =   0.000 deg,	R =   90.000 deg
};
P[323]{
   GP1:
	UF : 0, UT : 6,		CONFIG : 'N U T, 0, 0, 0',
	X =  145.739  mm,	Y =   -273.756  mm,	Z =   -324.061  mm,
	W =  90.000 deg,	P =   0.000 deg,	R =   90.000 deg
};
P[324]{
   GP1:
	UF : 0, UT : 6,		CONFIG : 'N U T, 0, 0, 0',
	X =  144.779  mm,	Y =   -273.933  mm,	Z =   -324.540  mm,
	W =  90.000 deg,	P =   0.000 deg,	R =   90.000 deg
};
P[325]{
   GP1:
	UF : 0, UT : 6,		CONFIG : 'N U T, 0, 0, 0',
	X =  143.574  mm,	Y =   -274.352  mm,	Z =   -322.371  mm,
	W =  90.000 deg,	P =   0.000 deg,	R =   90.000 deg
};
P[326]{
   GP1:
	UF : 0, UT : 6,		CONFIG : 'N U T, 0, 0, 0',
	X =  143.172  mm,	Y =   -275.465  mm,	Z =   -322.656  mm,
	W =  90.000 deg,	P =   0.000 deg,	R =   90.000 deg
};
P[327]{
   GP1:
	UF : 0, UT : 6,		CONFIG : 'N U T, 0, 0, 0',
	X =  142.457  mm,	Y =   -275.162  mm,	Z =   -314.680  mm,
	W =  90.000 deg,	P =   0.000 deg,	R =   90.000 deg
};
P[328]{
   GP1:
	UF : 0, UT : 6,		CONFIG : 'N U T, 0, 0, 0',
	X =  141.235  mm,	Y =   -276.007  mm,	Z =   -320.583  mm,
	W =  90.000 deg,	P =   0.000 deg,	R =   90.000 deg
};
P[329]{
   GP1:
	UF : 0, UT : 6,		CONFIG : 'N U T, 0, 0, 0',
	X =  139.778  mm,	Y =   -276.839  mm,	Z =   -323.425  mm,
	W =  90.000 deg,	P =   0.000 deg,	R =   90.000 deg
};
P[330]{
   GP1:
	UF : 0, UT : 6,		CONFIG : 'N U T, 0, 0, 0',
	X =  139.030  mm,	Y =   -277.352  mm,	Z =   -312.989  mm,
	W =  90.000 deg,	P =   0.000 deg,	R =   90.000 deg
};
P[331]{
   GP1:
	UF : 0, UT : 6,		CONFIG : 'N U T, 0, 0, 0',
	X =  137.952  mm,	Y =   -277.643  mm,	Z =   -321.278  mm,
	W =  90.000 deg,	P =   0.000 deg,	R =   90.000 deg
};
P[332]{
   GP1:
	UF : 0, UT : 6,		CONFIG : 'N U T, 0, 0, 0',
	X =  136.965  mm,	Y =   -278.708  mm,	Z =   -317.629  mm,
	W =  90.000 deg,	P =   0.000 deg,	R =   90.000 deg
};
P[333]{
   GP1:
	UF : 0, UT : 6,		CONFIG : 'N U T, 0, 0, 0',
	X =  135.994  mm,	Y =   -279.139  mm,	Z =   -309.930  mm,
	W =  90.000 deg,	P =   0.000 deg,	R =   90.000 deg
};
P[334]{
   GP1:
	UF : 0, UT : 6,		CONFIG : 'N U T, 0, 0, 0',
	X =  135.263  mm,	Y =   -279.963  mm,	Z =   -309.813  mm,
	W =  90.000 deg,	P =   0.000 deg,	R =   90.000 deg
};
P[335]{
   GP1:
	UF : 0, UT : 6,		CONFIG : 'N U T, 0, 0, 0',
	X =  134.116  mm,	Y =   -280.032  mm,	Z =   -326.781  mm,
	W =  90.000 deg,	P =   0.000 deg,	R =   90.000 deg
};
P[336]{
   GP1:
	UF : 0, UT : 6,		CONFIG : 'N U T, 0, 0, 0',
	X =  133.461  mm,	Y =   -280.388  mm,	Z =   -319.964  mm,
	W =  90.000 deg,	P =   0.000 deg,	R =   90.000 deg
};
P[337]{
   GP1:
	UF : 0, UT : 6,		CONFIG : 'N U T, 0, 0, 0',
	X =  132.576  mm,	Y =   -281.195  mm,	Z =   -315.012  mm,
	W =  90.000 deg,	P =   0.000 deg,	R =   90.000 deg
};
P[338]{
   GP1:
	UF : 0, UT : 6,		CONFIG : 'N U T, 0, 0, 0',
	X =  131.769  mm,	Y =   -281.560  mm,	Z =   -312.044  mm,
	W =  90.000 deg,	P =   0.000 deg,	R =   90.000 deg
};
P[339]{
   GP1:
	UF : 0, UT : 6,		CONFIG : 'N U T, 0, 0, 0',
	X =  131.139  mm,	Y =   -282.490  mm,	Z =   -324.044  mm,
	W =  90.000 deg,	P =   0.000 deg,	R =   90.000 deg
};
P[340]{
   GP1:
	UF : 0, UT : 6,		CONFIG : 'N U T, 0, 0, 0',
	X =  130.072  mm,	Y =   -282.234  mm,	Z =   -310.531  mm,
	W =  90.000 deg,	P =   0.000 deg,	R =   90.000 deg
};
P[341]{
   GP1:
	UF : 0, UT : 6,		CONFIG : 'N U T, 0, 0, 0',
	X =  129.157  mm,	Y =   -282.609  mm,	Z =   -314.274  mm,
	W =  90.000 deg,	P =   0.000 deg,	R =   90.000 deg
};
P[342]{
   GP1:
	UF : 0, UT : 6,		CONFIG : 'N U T, 0, 0, 0',
	X =  128.370  mm,	Y =   -283.586  mm,	Z =   -312.020  mm,
	W =  90.000 deg,	P =   0.000 deg,	R =   90.000 deg
};
P[343]{
   GP1:
	UF : 0, UT : 6,		CONFIG : 'N U T, 0, 0, 0',
	X =  127.589  mm,	Y =   -284.250  mm,	Z =   -319.858  mm,
	W =  90.000 deg,	P =   0.000 deg,	R =   90.000 deg
};
P[344]{
   GP1:
	UF : 0, UT : 6,		CONFIG : 'N U T, 0, 0, 0',
	X =  126.152  mm,	Y =   -284.494  mm,	Z =   -310.955  mm,
	W =  90.000 deg,	P =   0.000 deg,	R =   90.000 deg
};
P[345]{
   GP1:
	UF : 0, UT : 6,		CONFIG : 'N U T, 0, 0, 0',
	X =  125.723  mm,	Y =   -285.474  mm,	Z =   -309.903  mm,
	W =  90.000 deg,	P =   0.000 deg,	R =   90.000 deg
};
P[346]{
   GP1:
	UF : 0, UT : 6,		CONFIG : 'N U T, 0, 0, 0',
	X =  125.068  mm,	Y =   -285.757  mm,	Z =   -315.898  mm,
	W =  90.000 deg,	P =   0.000 deg,	R =   90.000 deg
};
P[347]{
   GP1:
	UF : 0, UT : 6,		CONFIG : 'N U T, 0, 0, 0',
	X =  125.092  mm,	Y =   -285.932  mm,	Z =   -327.312  mm,
	W =  90.000 deg,	P =   0.000 deg,	R =   90.000 deg
};
P[348]{
   GP1:
	UF : 0, UT : 6,		CONFIG : 'N U T, 0, 0, 0',
	X =  124.931  mm,	Y =   -285.680  mm,	Z =   -320.686  mm,
	W =  90.000 deg,	P =   0.000 deg,	R =   90.000 deg
};
P[349]{
   GP1:
	UF : 0, UT : 6,		CONFIG : 'N U T, 0, 0, 0',
	X =  124.761  mm,	Y =   -285.441  mm,	Z =   -325.611  mm,
	W =  90.000 deg,	P =   0.000 deg,	R =   90.000 deg
};
P[350]{
   GP1:
	UF : 0, UT : 6,		CONFIG : 'N U T, 0, 0, 0',
	X =  124.699  mm,	Y =   -286.144  mm,	Z =   -323.532  mm,
	W =  90.000 deg,	P =   0.000 deg,	R =   90.000 deg
};
P[351]{
   GP1:
	UF : 0, UT : 6,		CONFIG : 'N U T, 0, 0, 0',
	X =  124.243  mm,	Y =   -285.790  mm,	Z =   -322.352  mm,
	W =  90.000 deg,	P =   0.000 deg,	R =   90.000 deg
};
P[352]{
   GP1:
	UF : 0, UT : 6,		CONFIG : 'N U T, 0, 0, 0',
	X =  124.070  mm,	Y =   -285.713  mm,	Z =   -312.258  mm,
	W =  90.000 deg,	P =   0.000 deg,	R =   90.000 deg
};
P[353]{
   GP1:
	UF : 0, UT : 6,		CONFIG : 'N U T, 0, 0, 0',
	X =  124.173  mm,	Y =   -286.448  mm,	Z =   -324.680  mm,
	W =  90.000 deg,	P =   0.000 deg,	R =   90.000 deg
};
P[354]{
   GP1:
	UF : 0, UT : 6,		CONFIG : 'N U T, 0, 0, 0',
	X =  123.770  mm,	Y =   -285.969  mm,	Z =   -317.711  mm,
	W =  90.000 deg,	P =   0.000 deg,	R =   90.000 deg
};
P[355]{
   GP1:
	UF : 0, UT : 6,		CONFIG : 'N U T, 0, 0, 0',
	X =  123.819  mm,	Y =   -286.246  mm,	Z =   -313.172  mm,
	W =  90.000 deg,	P =   0.000 deg,	R =   90.000 deg
};
P[356]{
   GP1:
	UF : 0, UT : 6,		CONFIG : 'N U T, 0, 0, 0',
	X =  123.124  mm,	Y =   -286.169  mm,	Z =   -321.304  mm,
	W =  90.000 deg,	P =   0.000 deg,	R =   90.000 deg
};
P[357]{
   GP1:
	UF : 0, UT : 6,		CONFIG : 'N U T, 0, 0, 0',
	X =  123.054  mm,	Y =   -286.394  mm,	Z =   -319.367  mm,
	W =  90.000 deg,	P =   0.000 deg,	R =   90.000 deg
};
P[358]{
   GP1:
	UF : 0, UT : 6,		CONFIG : 'N U T, 0, 0, 0',
	X =  123.154  mm,	Y =   -286.634  mm,	Z =   -314.348  mm,
	W =  90.000 deg,	P =   0.000 deg,	R =   90.000 deg
};
P[359]{
   GP1:
	UF : 0, UT : 6,		CONFIG : 'N U T, 0, 0, 0',
	X =  123.216  mm,	Y =   -286.990  mm,	Z =   -321.318  mm,
	W =  90.000 deg,	P =   0.000 deg,	R =   90.000 deg
};
P[360]{
   GP1:
	UF : 0, UT : 6,		CONFIG : 'N U T, 0, 0, 0',
	X =  122.488  mm,	Y =   -286.848  mm,	Z =   -318.482  mm,
	W =  90.000 deg,	P =   0.000 deg,	R =   90.000 deg
};
P[361]{
   GP1:
	UF : 0, UT : 6,		CONFIG : 'N U T, 0, 0, 0',
	X =  122.626  mm,	Y =   -287.393  mm,	Z =   -327.120  mm,
	W =  90.000 deg,	P =   0.000 deg,	R =   90.000 deg
};
P[362]{
   GP1:
	UF : 0, UT : 6,		CONFIG : 'N U T, 0, 0, 0',
	X =  121.849  mm,	Y =   -287.268  mm,	Z =   -315.458  mm,
	W =  90.000 deg,	P =   0.000 deg,	R =   90.000 deg
};
P[363]{
   GP1:
	UF : 0, UT : 6,		CONFIG : 'N U T, 0, 0, 0',
	X =  121.664  mm,	Y =   -287.536  mm,	Z =   -319.029  mm,
	W =  90.000 deg,	P =   0.000 deg,	R =   90.000 deg
};
P[364]{
   GP1:
	UF : 0, UT : 6,		CONFIG : 'N U T, 0, 0, 0',
	X =  120.387  mm,	Y =   -287.803  mm,	Z =   -311.492  mm,
	W =  90.000 deg,	P =   0.000 deg,	R =   90.000 deg
};
P[365]{
   GP1:
	UF : 0, UT : 6,		CONFIG : 'N U T, 0, 0, 0',
	X =  120.623  mm,	Y =   -288.240  mm,	Z =   -323.842  mm,
	W =  90.000 deg,	P =   0.000 deg,	R =   90.000 deg
};
P[366]{
   GP1:
	UF : 0, UT : 6,		CONFIG : 'N U T, 0, 0, 0',
	X =  120.440  mm,	Y =   -288.610  mm,	Z =   -326.154  mm,
	W =  90.000 deg,	P =   0.000 deg,	R =   90.000 deg
};
P[367]{
   GP1:
	UF : 0, UT : 6,		CONFIG : 'N U T, 0, 0, 0',
	X =  119.788  mm,	Y =   -289.055  mm,	Z =   -324.797  mm,
	W =  90.000 deg,	P =   0.000 deg,	R =   90.000 deg
};
P[368]{
   GP1:
	UF : 0, UT : 6,		CONFIG : 'N U T, 0, 0, 0',
	X =  119.296  mm,	Y =   -288.427  mm,	Z =   -310.118  mm,
	W =  90.000 deg,	P =   0.000 deg,	R =   90.000 deg
};
P[369]{
   GP1:
	UF : 0, UT : 6,		CONFIG : 'N U T, 0, 0, 0',
	X =  118.943  mm,	Y =   -289.446  mm,	Z =   -322.181  mm,
	W =  90.000 deg,	P =   0.000 deg,	R =   90.000 deg
};
P[370]{
   GP1:
	UF : 0, UT : 6,		CONFIG : 'N U T, 0, 0, 0',
	X =  118.487  mm,	Y =   -289.144  mm,	Z =   -316.287  mm,
	W =  90.000 deg,	P =   0.000 deg,	R =   90.000 deg
};
P[371]{
   GP1:
	UF : 0, UT : 6,		CONFIG : 'N U T, 0, 0, 0',
	X =  118.000  mm,	Y =   -289.725  mm,	Z =   -327.861  mm,
	W =  90.000 deg,	P =   0.000 deg,	R =   90.000 deg
};
P[372]{
   GP1:
	UF : 0, UT : 6,		CONFIG : 'N U T, 0, 0, 0',
	X =  117.671  mm,	Y =   -289.465  mm,	Z =   -312.689  mm,
	W =  90.000 deg,	P =   0.000 deg,	R =   90.000 deg
};
P[373]{
   GP1:
	UF : 0, UT : 6,		CONFIG : 'N U T, 0, 0, 0',
	X =  116.989  mm,	Y =   -290.095  mm,	Z =   -312.441  mm,
	W =  90.000 deg,	P =   0.000 deg,	R =   90.000 deg
};
P[374]{
   GP1:
	UF : 0, UT : 6,		CONFIG : 'N U T, 0, 0, 0',
	X =  116.282  mm,	Y =   -290.487  mm,	Z =   -314.023  mm,
	W =  90.000 deg,	P =   0.000 deg,	R =   90.000 deg
};
P[375]{
   GP1:
	UF : 0, UT : 6,		CONFIG : 'N U T, 0, 0, 0',
	X =  116.070  mm,	Y =   -290.948  mm,	Z =   -316.558  mm,
	W =  90.000 deg,	P =   0.000 deg,	R =   90.000 deg
};
P[376]{
   GP1:
	UF : 0, UT : 6,		CONFIG : 'N U T, 0, 0, 0',
	X =  115.145  mm,	Y =   -291.038  mm,	Z =   -323.204  mm,
	W =  90.000 deg,	P =   0.000 deg,	R =   90.000 deg
};
P[377]{
   GP1:
	UF : 0, UT : 6,		CONFIG : 'N U T, 0, 0, 0',
	X =  115.104  mm,	Y =   -291.587  mm,	Z =   -311.068  mm,
	W =  90.000 deg,	P =   0.000 deg,	R =   90.000 deg
};
P[378]{
   GP1:
	UF : 0, UT : 6,		CONFIG : 'N U T, 0, 0, 0',
	X =  114.280  mm,	Y =   -291.465  mm,	Z =   -320.050  mm,
	W =  90.000 deg,	P =   0.000 deg,	R =   90.000 deg
};
P[379]{
   GP1:
	UF : 0, UT : 6,		CONFIG : 'N U T, 0, 0, 0',
	X =  113.515  mm,	Y =   -291.624  mm,	Z =   -325.401  mm,
	W =  90.000 deg,	P =   0.000 deg,	R =   90.000 deg
};
P[380]{
   GP1:
	UF : 0, UT : 6,		CONFIG : 'N U T, 0, 0, 0',
	X =  113.740  mm,	Y =   -292.147  mm,	Z =   -319.958  mm,
	W =  90.000 deg,	P =   0.000 deg,	R =   90.000 deg
};
P[381]{
   GP1:
	UF : 0, UT : 6,		CONFIG : 'N U T, 0, 0, 0',
	X =  113.319  mm,	Y =   -292.606  mm,	Z =   -312.037  mm,
	W =  90.000 deg,	P =   0.000 deg,	R =   90.000 deg
};
P[382]{
   GP1:
	UF : 0, UT : 6,		CONFIG : 'N U T, 0, 0, 0',
	X =  112.700  mm,	Y =   -292.425  mm,	Z =   -325.777  mm,
	W =  90.000 deg,	P =   0.000 deg,	R =   90.000 deg
};
P[383]{
   GP1:
	UF : 0, UT : 6,		CONFIG : 'N U T, 0, 0, 0',
	X =  111.579  mm,	Y =   -293.271  mm,	Z =   -311.321  mm,
	W =  90.000 deg,	P =   0.000 deg,	R =   90.000 deg
};
P[384]{
   GP1:
	UF : 0, UT : 6,		CONFIG : 'N U T, 0, 0, 0',
	X =  111.546  mm,	Y =   -293.839  mm,	Z =   -321.038  mm,
	W =  90.000 deg,	P =   0.000 deg,	R =   90.000 deg
};
P[385]{
   GP1:
	UF : 0, UT : 6,		CONFIG : 'N U T, 0, 0, 0',
	X =  110.615  mm,	Y =   -293.706  mm,	Z =   -317.393  mm,
	W =  90.000 deg,	P =   0.000 deg,	R =   90.000 deg
};
P[386]{
   GP1:
	UF : 0, UT : 6,		CONFIG : 'N U T, 0, 0, 0',
	X =  110.268  mm,	Y =   -294.229  mm,	Z =   -324.946  mm,
	W =  90.000 deg,	P =   0.000 deg,	R =   90.000 deg
};
P[387]{
   GP1:
	UF : 0, UT : 6,		CONFIG : 'N U T, 0, 0, 0',
	X =  108.959  mm,	Y =   -294.445  mm,	Z =   -311.843  mm,
	W =  90.000 deg,	P =   0.000 deg,	R =   90.000 deg
};
P[388]{
   GP1:
	UF : 0, UT : 6,		CONFIG : 'N U T, 0, 0, 0',
	X =  108.961  mm,	Y =   -295.077  mm,	Z =   -314.775  mm,
	W =  90.000 deg,	P =   0.000 deg,	R =   90.000 deg
};
P[389]{
   GP1:
	UF : 0, UT : 6,		CONFIG : 'N U T, 0, 0, 0',
	X =  107.851  mm,	Y =   -294.964  mm,	Z =   -324.794  mm,
	W =  90.000 deg,	P =   0.000 deg,	R =   90.000 deg
};
P[390]{
   GP1:
	UF : 0, UT : 6,		CONFIG : 'N U T, 0, 0, 0',
	X =  108.161  mm,	Y =   -295.757  mm,	Z =   -324.638  mm,
	W =  90.000 deg,	P =   0.000 deg,	R =   90.000 deg
};
P[391]{
   GP1:
	UF : 0, UT : 6,		CONFIG : 'N U T, 0, 0, 0',
	X =  107.638  mm,	Y =   -295.591  mm,	Z =   -315.039  mm,
	W =  90.000 deg,	P =   0.000 deg,	R =   90.000 deg
};
P[392]{
   GP1:
	UF : 0, UT : 6,		CONFIG : 'N U T, 0, 0, 0',
	X =  107.077  mm,	Y =   -295.404  mm,	Z =   -326.572  mm,
	W =  90.000 deg,	P =   0.000 deg,	R =   90.000 deg
};
P[393]{
   GP1:
	UF : 0, UT : 6,		CONFIG : 'N U T, 0, 0, 0',
	X =  106.802  mm,	Y =   -296.362  mm,	Z =   -312.153  mm,
	W =  90.000 deg,	P =   0.000 deg,	R =   90.000 deg
};
P[394]{
   GP1:
	UF : 0, UT : 6,		CONFIG : 'N U T, 0, 0, 0',
	X =  106.166  mm,	Y =   -296.127  mm,	Z =   -317.068  mm,
	W =  90.000 deg,	P =   0.000 deg,	R =   90.000 deg
};
P[395]{
   GP1:
	UF : 0, UT : 6,		CONFIG : 'N U T, 0, 0, 0',
	X =  105.472  mm,	Y =   -296.373  mm,	Z =   -321.590  mm,
	W =  90.000 deg,	P =   0.000 deg,	R =   90.000 deg
};
P[396]{
   GP1:
	UF : 0, UT : 6,		CONFIG : 'N U T, 0, 0, 0',
	X =  105.506  mm,	Y =   -297.304  mm,	Z =   -323.017  mm,
	W =  90.000 deg,	P =   0.000 deg,	R =   90.000 deg
};
P[397]{
   GP1:
	UF : 0, UT : 6,		CONFIG : 'N U T, 0, 0, 0',
	X =  104.898  mm,	Y =   -297.180  mm,	Z =   -314.230  mm,
	W =  90.000 deg,	P =   0.000 deg,	R =   90.000 deg
};
P[398]{
   GP1:
	UF : 0, UT : 6,		CONFIG : 'N U T, 0, 0, 0',
	X =  104.041  mm,	Y =   -297.404  mm,	Z =   -327.657  mm,
	W =  90.000 deg,	P =   0.000 deg,	R =   90.000 deg
};
P[399]{
   GP1:
	UF : 0, UT : 6,		CONFIG : 'N U T, 0, 0, 0',
	X =  103.867  mm,	Y =   -297.957  mm,	Z =   -318.669  mm,
	W =  90.000 deg,	P =   0.000 deg,	R =   90.000 deg
};
P[400]{
   GP1:
	UF : 0, UT : 6,		CONFIG : 'N U T, 0, 0, 0',
	X =  103.214  mm,	Y =   -297.538  mm,	Z =   -324.099  mm,
	W =  90.000 deg,	P =   0.000 deg,	R =   90.000 deg
};
P[401]{
   GP1:
	UF : 0, UT : 6,		CONFIG : 'N U T, 0, 0, 0',
	X =  103.145  mm,	Y =   -298.401  mm,	Z =   -316.025  mm,
	W =  90.000 deg,	P =   0.000 deg,	R =   90.000 deg
};
P[402]{
   GP1:
	UF : 0, UT : 6,		CONFIG : 'N U T, 0, 0, 0',
	X =  102.179  mm,	Y =   -298.477  mm,	Z =   -326.155  mm,
	W =  90.000 deg,	P =   0.000 deg,	R =   90.000 deg
};
P[403]{
   GP1:
	UF : 0, UT : 6,		CONFIG : 'N U T, 0, 0, 0',
	X =  102.123  mm,	Y =   -299.241  mm,	Z =   -324.346  mm,
	W =  90.000 deg,	P =   0.000 deg,	R =   90.000 deg
};
P[404]{
   GP1:
	UF : 0, UT : 6,		CONFIG : 'N U T, 0, 0, 0',
	X =  101.634  mm,	Y =   -299.115  mm,	Z =   -317.204  mm,
	W =  90.000 deg,	P =   0.000 deg,	R =   90.000 deg
};
P[405]{
   GP1:
	UF : 0, UT : 6,		CONFIG : 'N U T, 0, 0, 0',
	X =  100.604  mm,	Y =   -299.421  mm,	Z =   -327.287  mm,
	W =  90.000 deg,	P =   0.000 deg,	R =   90.000 deg
};
P[406]{
   GP1:
	UF : 0, UT : 6,		CONFIG : 'N U T, 0, 0, 0',
	X =  100.339  mm,	Y =   -300.028  mm,	Z =   -315.838  mm,
	W =  90.000 deg,	P =   0.000 deg,	R =   90.000 deg
};
P[407]{
   GP1:
	UF : 0, UT : 6,		CONFIG : 'N U T, 0, 0, 0',
	X =  99.550  mm,	Y =   -300.023  mm,	Z =   -326.447  mm,
	W =  90.000 deg,	P =   0.000 deg,	R =   90.000 deg
};
P[408]{
   GP1:
	UF : 0, UT : 6,		CONFIG : 'N U T, 0, 0, 0',
	X =  99.683  mm,	Y =   -300.640  mm,	Z =   -324.924  mm,
	W =  90.000 deg,	P =   0.000 deg,	R =   90.000 deg
};
P[409]{
   GP1:
	UF : 0, UT : 6,		CONFIG : 'N U T, 0, 0, 0',
	X =  99.164  mm,	Y =   -300.588  mm,	Z =   -326.808  mm,
	W =  90.000 deg,	P =   0.000 deg,	R =   90.000 deg
};
P[410]{
   GP1:
	UF : 0, UT : 6,		CONFIG : 'N U T, 0, 0, 0',
	X =  98.683  mm,	Y =   -300.395  mm,	Z =   -313.181  mm,
	W =  90.000 deg,	P =   0.000 deg,	R =   90.000 deg
};
P[411]{
   GP1:
	UF : 0, UT : 6,		CONFIG : 'N U T, 0, 0, 0',
	X =  98.177  mm,	Y =   -301.534  mm,	Z =   -323.604  mm,
	W =  90.000 deg,	P =   0.000 deg,	R =   90.000 deg
};
P[412]{
   GP1:
	UF : 0, UT : 6,		CONFIG : 'N U T, 0, 0, 0',
	X =  97.652  mm,	Y =   -301.231  mm,	Z =   -315.302  mm,
	W =  90.000 deg,	P =   0.000 deg,	R =   90.000 deg
};
P[413]{
   GP1:
	UF : 0, UT : 6,		CONFIG : 'N U T, 0, 0, 0',
	X =  97.046  mm,	Y =   -301.314  mm,	Z =   -310.430  mm,
	W =  90.000 deg,	P =   0.000 deg,	R =   90.000 deg
};
P[414]{
   GP1:
	UF : 0, UT : 6,		CONFIG : 'N U T, 0, 0, 0',
	X =  96.850  mm,	Y =   -301.987  mm,	Z =   -319.869  mm,
	W =  90.000 deg,	P =   0.000 deg,	R =   90.000 deg
};
P[415]{
   GP1:
	UF : 0, UT : 6,		CONFIG : 'N U T, 0, 0, 0',
	X =  96.235  mm,	Y =   -301.859  mm,	Z =   -317.697  mm,
	W =  90.000 deg,	P =   0.000 deg,	R =   90.000 deg
};
P[416]{
   GP1:
	UF : 0, UT : 6,		CONFIG : 'N U T, 0, 0, 0',
	X =  96.241  mm,	Y =   -302.200  mm,	Z =   -317.003  mm,
	W =  90.000 deg,	P =   0.000 deg,	R =   90.000 deg
};
P[417]{
   GP1:
	UF : 0, UT : 6,		CONFIG : 'N U T, 0, 0, 0',
	X =  95.516  mm,	Y =   -301.987  mm,	Z =   -321.449  mm,
	W =  90.000 deg,	P =   0.000 deg,	R =   90.000 deg
};
P[418]{
   GP1:
	UF : 0, UT : 6,		CONFIG : 'N U T, 0, 0, 0',
	X =  95.720  mm,	Y =   -302.706  mm,	Z =   -315.209  mm,
	W =  90.000 deg,	P =   0.000 deg,	R =   90.000 deg
};
P[419]{
   GP1:
	UF : 0, UT : 6,		CONFIG : 'N U T, 0, 0, 0',
	X =  95.349  mm,	Y =   -302.639  mm,	Z =   -310.140  mm,
	W =  90.000 deg,	P =   0.000 deg,	R =   90.000 deg
};
P[420]{
   GP1:
	UF : 0, UT : 6,		CONFIG : 'N U T, 0, 0, 0',
	X =  94.560  mm,	Y =   -302.843  mm,	Z =   -318.549  mm,
	W =  90.000 deg,	P =   0.000 deg,	R =   90.000 deg
};
P[421]{
   GP1:
	UF : 0, UT : 6,		CONFIG : 'N U T, 0, 0, 0',
	X =  94.439  mm,	Y =   -302.642  mm,	Z =   -324.089  mm,
	W =  90.000 deg,	P =   0.000 deg,	R =   90.000 deg
};
P[422]{
   GP1:
	UF : 0, UT : 6,		CONFIG : 'N U T, 0, 0, 0',
	X =  94.507  mm,	Y =   -303.246  mm,	Z =   -320.243  mm,
	W =  90.000 deg,	P =   0.000 deg,	R =   90.000 deg
};
P[423]{
   GP1:
	UF : 0, UT : 6,		CONFIG : 'N U T, 0, 0, 0',
	X =  94.509  mm,	Y =   -303.687  mm,	Z =   -322.063  mm,
	W =  90.000 deg,	P =   0.000 deg,	R =   90.000 deg
};
P[424]{
   GP1:
	UF : 0, UT : 6,		CONFIG : 'N U T, 0, 0, 0',
	X =  93.529  mm,	Y =   -303.114  mm,	Z =   -318.902  mm,
	W =  90.000 deg,	P =   0.000 deg,	R =   90.000 deg
};
P[425]{
   GP1:
	UF : 0, UT : 6,		CONFIG : 'N U T, 0, 0, 0',
	X =  93.557  mm,	Y =   -303.319  mm,	Z =   -310.362  mm,
	W =  90.000 deg,	P =   0.000 deg,	R =   90.000 deg
};
P[426]{
   GP1:
	UF : 0, UT : 6,		CONFIG : 'N U T, 0, 0, 0',
	X =  93.664  mm,	Y =   -303.617  mm,	Z =   -311.970  mm,
	W =  90.000 deg,	P =   0.000 deg,	R =   90.000 deg
};
P[427]{
   GP1:
	UF : 0, UT : 6,		CONFIG : 'N U T, 0, 0, 0',
	X =  93.856  mm,	Y =   -304.068  mm,	Z =   -320.152  mm,
	W =  90.000 deg,	P =   0.000 deg,	R =   90.000 deg
};
P[428]{
   GP1:
	UF : 0, UT : 6,		CONFIG : 'N U T, 0, 0, 0',
	X =  93.142  mm,	Y =   -304.156  mm,	Z =   -317.392  mm,
	W =  90.000 deg,	P =   0.000 deg,	R =   90.000 deg
};
P[429]{
   GP1:
	UF : 0, UT : 6,		CONFIG : 'N U T, 0, 0, 0',
	X =  92.699  mm,	Y =   -303.841  mm,	Z =   -311.772  mm,
	W =  90.000 deg,	P =   0.000 deg,	R =   90.000 deg
};
P[430]{
   GP1:
	UF : 0, UT : 6,		CONFIG : 'N U T, 0, 0, 0',
	X =  92.832  mm,	Y =   -304.138  mm,	Z =   -314.028  mm,
	W =  90.000 deg,	P =   0.000 deg,	R =   90.000 deg
};
P[431]{
   GP1:
	UF : 0, UT : 6,		CONFIG : 'N U T, 0, 0, 0',
	X =  92.337  mm,	Y =   -303.898  mm,	Z =   -325.183  mm,
	W =  90.000 deg,	P =   0.000 deg,	R =   90.000 deg
};
P[432]{
   GP1:
	UF : 0, UT : 6,		CONFIG : 'N U T, 0, 0, 0',
	X =  92.337  mm,	Y =   -304.720  mm,	Z =   -312.325  mm,
	W =  90.000 deg,	P =   0.000 deg,	R =   90.000 deg
};
P[433]{
   GP1:
	UF : 0, UT : 6,		CONFIG : 'N U T, 0, 0, 0',
	X =  91.891  mm,	Y =   -304.305  mm,	Z =   -311.900  mm,
	W =  90.000 deg,	P =   0.000 deg,	R =   90.000 deg
};
P[434]{
   GP1:
	UF : 0, UT : 6,		CONFIG : 'N U T, 0, 0, 0',
	X =  91.972  mm,	Y =   -304.486  mm,	Z =   -316.898  mm,
	W =  90.000 deg,	P =   0.000 deg,	R =   90.000 deg
};
P[435]{
   GP1:
	UF : 0, UT : 6,		CONFIG : 'N U T, 0, 0, 0',
	X =  91.621  mm,	Y =   -304.353  mm,	Z =   -323.567  mm,
	W =  90.000 deg,	P =   0.000 deg,	R =   90.000 deg
};
P[436]{
   GP1:
	UF : 0, UT : 6,		CONFIG : 'N U T, 0, 0, 0',
	X =  91.731  mm,	Y =   -304.961  mm,	Z =   -317.212  mm,
	W =  90.000 deg,	P =   0.000 deg,	R =   90.000 deg
};
P[437]{
   GP1:
	UF : 0, UT : 6,		CONFIG : 'N U T, 0, 0, 0',
	X =  91.224  mm,	Y =   -304.608  mm,	Z =   -322.031  mm,
	W =  90.000 deg,	P =   0.000 deg,	R =   90.000 deg
};
P[438]{
   GP1:
	UF : 0, UT : 6,		CONFIG : 'N U T, 0, 0, 0',
	X =  91.107  mm,	Y =   -304.911  mm,	Z =   -327.091  mm,
	W =  90.000 deg,	P =   0.000 deg,	R =   90.000 deg
};
P[439]{
   GP1:
	UF : 0, UT : 6,		CONFIG : 'N U T, 0, 0, 0',
	X =  91.019  mm,	Y =   -304.870  mm,	Z =   -317.005  mm,
	W =  90.000 deg,	P =   0.000 deg,	R =   90.000 deg
};
P[440]{
   GP1:
	UF : 0, UT : 6,		CONFIG : 'N U T, 0, 0, 0',
	X =  90.892  mm,	Y =   -305.335  mm,	Z =   -320.063  mm,
	W =  90.000 deg,	P =   0.000 deg,	R =   90.000 deg
};
P[441]{
   GP1:
	UF : 0, UT : 6,		CONFIG : 'N U T, 0, 0, 0',
	X =  90.967  mm,	Y =   -305.584  mm,	Z =   -322.766  mm,
	W =  90.000 deg,	P =   0.000 deg,	R =   90.000 deg
};
P[442]{
   GP1:
	UF : 0, UT : 6,		CONFIG : 'N U T, 0, 0, 0',
	X =  90.455  mm,	Y =   -305.341  mm,	Z =   -317.648  mm,
	W =  90.000 deg,	P =   0.000 deg,	R =   90.000 deg
};
P[443]{
   GP1:
	UF : 0, UT : 6,		CONFIG : 'N U T, 0, 0, 0',
	X =  90.383  mm,	Y =   -305.319  mm,	Z =   -327.801  mm,
	W =  90.000 deg,	P =   0.000 deg,	R =   90.000 deg
};
P[444]{
   GP1:
	UF : 0, UT : 6,		CONFIG : 'N U T, 0, 0, 0',
	X =  90.414  mm,	Y =   -305.560  mm,	Z =   -316.949  mm,
	W =  90.000 deg,	P =   0.000 deg,	R =   90.000 deg
};
P[445]{
   GP1:
	UF : 0, UT : 6,		CONFIG : 'N U T, 0, 0, 0',
	X =  90.292  mm,	Y =   -306.017  mm,	Z =   -324.070  mm,
	W =  90.000 deg,	P =   0.000 deg,	R =   90.000 deg
};
P[446]{
   GP1:
	UF : 0, UT : 6,		CONFIG : 'N U T, 0, 0, 0',
	X =  89.646  mm,	Y =   -306.021  mm,	Z =   -316.841  mm,
	W =  90.000 deg,	P =   0.000 deg,	R =   90.000 deg
};
P[447]{
   GP1:
	UF : 0, UT : 6,		CONFIG : 'N U T, 0, 0, 0',
	X =  89.620  mm,	Y =   -306.388  mm,	Z =   -321.204  mm,
	W =  90.000 deg,	P =   0.000 deg,	R =   90.000 deg
};
P[448]{
   GP1:
	UF : 0, UT : 6,		CONFIG : 'N U T, 0, 0, 0',
	X =  89.459  mm,	Y =   -306.342  mm,	Z =   -314.694  mm,
	W =  90.000 deg,	P =   0.000 deg,	R =   90.000 deg
};
P[449]{
   GP1:
	UF : 0, UT : 6,		CONFIG : 'N U T, 0, 0, 0',
	X =  89.258  mm,	Y =   -306.256  mm,	Z =   -318.643  mm,
	W =  90.000 deg,	P =   0.000 deg,	R =   90.000 deg
};
P[450]{
   GP1:
	UF : 0, UT : 6,		CONFIG : 'N U T, 0, 0, 0',
	X =  88.865  mm,	Y =   -306.790  mm,	Z =   -321.772  mm,
	W =  90.000 deg,	P =   0.000 deg,	R =   90.000 deg
};
P[451]{
   GP1:
	UF : 0, UT : 6,		CONFIG : 'N U T, 0, 0, 0',
	X =  88.796  mm,	Y =   -306.940  mm,	Z =   -324.200  mm,
	W =  90.000 deg,	P =   0.000 deg,	R =   90.000 deg
};
P[452]{
   GP1:
	UF : 0, UT : 6,		CONFIG : 'N U T, 0, 0, 0',
	X =  88.692  mm,	Y =   -306.868  mm,	Z =   -322.787  mm,
	W =  90.000 deg,	P =   0.000 deg,	R =   90.000 deg
};
P[453]{
   GP1:
	UF : 0, UT : 6,		CONFIG : 'N U T, 0, 0, 0',
	X =  88.281  mm,	Y =   -306.318  mm,	Z =   -321.216  mm,
	W =  90.000 deg,	P =   0.000 deg,	R =   90.000 deg
};
P[454]{
   GP1:
	UF : 0, UT : 6,		CONFIG : 'N U T, 0, 0, 0',
	X =  88.246  mm,	Y =   -307.189  mm,	Z =   -327.163  mm,
	W =  90.000 deg,	P =   0.000 deg,	R =   90.000 deg
};
P[455]{
   GP1:
	UF : 0, UT : 6,		CONFIG : 'N U T, 0, 0, 0',
	X =  87.578  mm,	Y =   -307.103  mm,	Z =   -309.805  mm,
	W =  90.000 deg,	P =   0.000 deg,	R =   90.000 deg
};
P[456]{
   GP1:
	UF : 0, UT : 6,		CONFIG : 'N U T, 0, 0, 0',
	X =  86.745  mm,	Y =   -307.814  mm,	Z =   -323.570  mm,
	W =  90.000 deg,	P =   0.000 deg,	R =   90.000 deg
};
P[457]{
   GP1:
	UF : 0, UT : 6,		CONFIG : 'N U T, 0, 0, 0',
	X =  85.957  mm,	Y =   -307.998  mm,	Z =   -313.982  mm,
	W =  90.000 deg,	P =   0.000 deg,	R =   90.000 deg
};
P[458]{
   GP1:
	UF : 0, UT : 6,		CONFIG : 'N U T, 0, 0, 0',
	X =  85.061  mm,	Y =   -308.635  mm,	Z =   -315.886  mm,
	W =  90.000 deg,	P =   0.000 deg,	R =   90.000 deg
};
P[459]{
   GP1:
	UF : 0, UT : 6,		CONFIG : 'N U T, 0, 0, 0',
	X =  83.337  mm,	Y =   -309.167  mm,	Z =   -322.331  mm,
	W =  90.000 deg,	P =   0.000 deg,	R =   90.000 deg
};
P[460]{
   GP1:
	UF : 0, UT : 6,		CONFIG : 'N U T, 0, 0, 0',
	X =  82.559  mm,	Y =   -310.062  mm,	Z =   -312.873  mm,
	W =  90.000 deg,	P =   0.000 deg,	R =   90.000 deg
};
P[461]{
   GP1:
	UF : 0, UT : 6,		CONFIG : 'N U T, 0, 0, 0',
	X =  82.072  mm,	Y =   -310.812  mm,	Z =   -323.800  mm,
	W =  90.000 deg,	P =   0.000 deg,	R =   90.000 deg
};
P[462]{
   GP1:
	UF : 0, UT : 6,		CONFIG : 'N U T, 0, 0, 0',
	X =  80.836  mm,	Y =   -311.312  mm,	Z =   -316.029  mm,
	W =  90.000 deg,	P =   0.000 deg,	R =   90.000 deg
};
P[463]{
   GP1:
	UF : 0, UT : 6,		CONFIG : 'N U T, 0, 0, 0',
	X =  78.315  mm,	Y =   -312.443  mm,	Z =   -320.592  mm,
	W =  90.000 deg,	P =   0.000 deg,	R =   90.000 deg
};
P[464]{
   GP1:
	UF : 0, UT : 6,		CONFIG : 'N U T, 0, 0, 0',
	X =  77.255  mm,	Y =   -313.601  mm,	Z =   -322.468  mm,
	W =  90.000 deg,	P =   0.000 deg,	R =   90.000 deg
};
P[465]{
   GP1:
	UF : 0, UT : 6,		CONFIG : 'N U T, 0, 0, 0',
	X =  76.171  mm,	Y =   -313.525  mm,	Z =   -325.147  mm,
	W =  90.000 deg,	P =   0.000 deg,	R =   90.000 deg
};
P[466]{
   GP1:
	UF : 0, UT : 6,		CONFIG : 'N U T, 0, 0, 0',
	X =  75.705  mm,	Y =   -314.110  mm,	Z =   -326.346  mm,
	W =  90.000 deg,	P =   0.000 deg,	R =   90.000 deg
};
P[467]{
   GP1:
	UF : 0, UT : 6,		CONFIG : 'N U T, 0, 0, 0',
	X =  74.850  mm,	Y =   -314.523  mm,	Z =   -315.082  mm,
	W =  90.000 deg,	P =   0.000 deg,	R =   90.000 deg
};
P[468]{
   GP1:
	UF : 0, UT : 6,		CONFIG : 'N U T, 0, 0, 0',
	X =  73.955  mm,	Y =   -314.834  mm,	Z =   -323.620  mm,
	W =  90.000 deg,	P =   0.000 deg,	R =   90.000 deg
};
P[469]{
   GP1:
	UF : 0, UT : 6,		CONFIG : 'N U T, 0, 0, 0',
	X =  73.083  mm,	Y =   -315.362  mm,	Z =   -320.266  mm,
	W =  90.000 deg,	P =   0.000 deg,	R =   90.000 deg
};
P[470]{
   GP1:
	UF : 0, UT : 6,		CONFIG : 'N U T, 0, 0, 0',
	X =  72.125  mm,	Y =   -315.827  mm,	Z =   -325.926  mm,
	W =  90.000 deg,	P =   0.000 deg,	R =   90.000 deg
};
P[471]{
   GP1:
	UF : 0, UT : 6,		CONFIG : 'N U T, 0, 0, 0',
	X =  71.187  mm,	Y =   -316.044  mm,	Z =   -323.385  mm,
	W =  90.000 deg,	P =   0.000 deg,	R =   90.000 deg
};
P[472]{
   GP1:
	UF : 0, UT : 6,		CONFIG : 'N U T, 0, 0, 0',
	X =  70.848  mm,	Y =   -317.048  mm,	Z =   -316.667  mm,
	W =  90.000 deg,	P =   0.000 deg,	R =   90.000 deg
};
P[473]{
   GP1:
	UF : 0, UT : 6,		CONFIG : 'N U T, 0, 0, 0',
	X =  69.295  mm,	Y =   -317.427  mm,	Z =   -318.747  mm,
	W =  90.000 deg,	P =   0.000 deg,	R =   90.000 deg
};
P[474]{
   GP1:
	UF : 0, UT : 6,		CONFIG : 'N U T, 0, 0, 0',
	X =  68.171  mm,	Y =   -317.851  mm,	Z =   -324.440  mm,
	W =  90.000 deg,	P =   0.000 deg,	R =   90.000 deg
};
P[475]{
   GP1:
	UF : 0, UT : 6,		CONFIG : 'N U T, 0, 0, 0',
	X =  67.831  mm,	Y =   -318.536  mm,	Z =   -311.985  mm,
	W =  90.000 deg,	P =   0.000 deg,	R =   90.000 deg
};
P[476]{
   GP1:
	UF : 0, UT : 6,		CONFIG : 'N U T, 0, 0, 0',
	X =  66.795  mm,	Y =   -319.174  mm,	Z =   -315.053  mm,
	W =  90.000 deg,	P =   0.000 deg,	R =   90.000 deg
};
P[477]{
   GP1:
	UF : 0, UT : 6,		CONFIG : 'N U T, 0, 0, 0',
	X =  65.515  mm,	Y =   -319.651  mm,	Z =   -326.317  mm,
	W =  90.000 deg,	P =   0.000 deg,	R =   90.000 deg
};
P[478]{
   GP1:
	UF : 0, UT : 6,		CONFIG : 'N U T, 0, 0, 0',
	X =  64.469  mm,	Y =   -320.629  mm,	Z =   -325.935  mm,
	W =  90.000 deg,	P =   0.000 deg,	R =   90.000 deg
};
P[479]{
   GP1:
	UF : 0, UT : 6,		CONFIG : 'N U T, 0, 0, 0',
	X =  63.291  mm,	Y =   -320.760  mm,	Z =   -309.929  mm,
	W =  90.000 deg,	P =   0.000 deg,	R =   90.000 deg
};
P[480]{
   GP1:
	UF : 0, UT : 6,		CONFIG : 'N U T, 0, 0, 0',
	X =  70.879  mm,	Y =   -334.019  mm,	Z =   -322.479  mm,
	W =  90.000 deg,	P =   0.000 deg,	R =   90.000 deg
};
P[481]{
   GP1:
	UF : 0, UT : 6,		CONFIG : 'N U T, 0, 0, 0',
	X =  72.024  mm,	Y =   -333.189  mm,	Z =   -322.103  mm,
	W =  90.000 deg,	P =   0.000 deg,	R =   90.000 deg
};
P[482]{
   GP1:
	UF : 0, UT : 6,		CONFIG : 'N U T, 0, 0, 0',
	X =  72.726  mm,	Y =   -332.635  mm,	Z =   -323.884  mm,
	W =  90.000 deg,	P =   0.000 deg,	R =   90.000 deg
};
P[483]{
   GP1:
	UF : 0, UT : 6,		CONFIG : 'N U T, 0, 0, 0',
	X =  73.561  mm,	Y =   -332.589  mm,	Z =   -318.130  mm,
	W =  90.000 deg,	P =   0.000 deg,	R =   90.000 deg
};
P[484]{
   GP1:
	UF : 0, UT : 6,		CONFIG : 'N U T, 0, 0, 0',
	X =  74.461  mm,	Y =   -332.054  mm,	Z =   -315.948  mm,
	W =  90.000 deg,	P =   0.000 deg,	R =   90.000 deg
};
P[485]{
   GP1:
	UF : 0, UT : 6,		CONFIG : 'N U T, 0, 0, 0',
	X =  74.954  mm,	Y =   -331.223  mm,	Z =   -319.189  mm,
	W =  90.000 deg,	P =   0.000 deg,	R =   90.000 deg
};
P[486]{
   GP1:
	UF : 0, UT : 6,		CONFIG : 'N U T, 0, 0, 0',
	X =  76.142  mm,	Y =   -331.196  mm,	Z =   -322.437  mm,
	W =  90.000 deg,	P =   0.000 deg,	R =   90.000 deg
};
P[487]{
   GP1:
	UF : 0, UT : 6,		CONFIG : 'N U T, 0, 0, 0',
	X =  76.824  mm,	Y =   -330.459  mm,	Z =   -325.046  mm,
	W =  90.000 deg,	P =   0.000 deg,	R =   90.000 deg
};
P[488]{
   GP1:
	UF : 0, UT : 6,		CONFIG : 'N U T, 0, 0, 0',
	X =  77.820  mm,	Y =   -330.270  mm,	Z =   -318.553  mm,
	W =  90.000 deg,	P =   0.000 deg,	R =   90.000 deg
};
P[489]{
   GP1:
	UF : 0, UT : 6,		CONFIG : 'N U T, 0, 0, 0',
	X =  78.789  mm,	Y =   -329.806  mm,	Z =   -312.479  mm,
	W =  90.000 deg,	P =   0.000 deg,	R =   90.000 deg
};
P[490]{
   GP1:
	UF : 0, UT : 6,		CONFIG : 'N U T, 0, 0, 0',
	X =  79.575  mm,	Y =   -329.571  mm,	Z =   -324.763  mm,
	W =  90.000 deg,	P =   0.000 deg,	R =   90.000 deg
};
P[491]{
   GP1:
	UF : 0, UT : 6,		CONFIG : 'N U T, 0, 0, 0',
	X =  80.164  mm,	Y =   -328.716  mm,	Z =   -311.952  mm,
	W =  90.000 deg,	P =   0.000 deg,	R =   90.000 deg
};
P[492]{
   GP1:
	UF : 0, UT : 6,		CONFIG : 'N U T, 0, 0, 0',
	X =  81.306  mm,	Y =   -327.599  mm,	Z =   -318.417  mm,
	W =  90.000 deg,	P =   0.000 deg,	R =   90.000 deg
};
P[493]{
   GP1:
	UF : 0, UT : 6,		CONFIG : 'N U T, 0, 0, 0',
	X =  82.304  mm,	Y =   -327.581  mm,	Z =   -320.262  mm,
	W =  90.000 deg,	P =   0.000 deg,	R =   90.000 deg
};
P[494]{
   GP1:
	UF : 0, UT : 6,		CONFIG : 'N U T, 0, 0, 0',
	X =  83.183  mm,	Y =   -326.891  mm,	Z =   -325.242  mm,
	W =  90.000 deg,	P =   0.000 deg,	R =   90.000 deg
};
P[495]{
   GP1:
	UF : 0, UT : 6,		CONFIG : 'N U T, 0, 0, 0',
	X =  84.898  mm,	Y =   -326.283  mm,	Z =   -312.442  mm,
	W =  90.000 deg,	P =   0.000 deg,	R =   90.000 deg
};
P[496]{
   GP1:
	UF : 0, UT : 6,		CONFIG : 'N U T, 0, 0, 0',
	X =  85.872  mm,	Y =   -325.124  mm,	Z =   -319.072  mm,
	W =  90.000 deg,	P =   0.000 deg,	R =   90.000 deg
};
P[497]{
   GP1:
	UF : 0, UT : 6,		CONFIG : 'N U T, 0, 0, 0',
	X =  85.942  mm,	Y =   -325.245  mm,	Z =   -322.952  mm,
	W =  90.000 deg,	P =   0.000 deg,	R =   90.000 deg
};
P[498]{
   GP1:
	UF : 0, UT : 6,		CONFIG : 'N U T, 0, 0, 0',
	X =  85.962  mm,	Y =   -325.280  mm,	Z =   -327.321  mm,
	W =  90.000 deg,	P =   0.000 deg,	R =   90.000 deg
};
P[499]{
   GP1:
	UF : 0, UT : 6,		CONFIG : 'N U T, 0, 0, 0',
	X =  85.974  mm,	Y =   -325.301  mm,	Z =   -322.942  mm,
	W =  90.000 deg,	P =   0.000 deg,	R =   90.000 deg
};
P[500]{
   GP1:
	UF : 0, UT : 6,		CONFIG : 'N U T, 0, 0, 0',
	X =  85.979  mm,	Y =   -325.310  mm,	Z =   -321.277  mm,
	W =  90.000 deg,	P =   0.000 deg,	R =   90.000 deg
};
P[501]{
   GP1:
	UF : 0, UT : 6,		CONFIG : 'N U T, 0, 0, 0',
	X =  86.076  mm,	Y =   -325.478  mm,	Z =   -320.153  mm,
	W =  90.000 deg,	P =   0.000 deg,	R =   90.000 deg
};
P[502]{
   GP1:
	UF : 0, UT : 6,		CONFIG : 'N U T, 0, 0, 0',
	X =  86.083  mm,	Y =   -325.490  mm,	Z =   -320.938  mm,
	W =  90.000 deg,	P =   0.000 deg,	R =   90.000 deg
};
P[503]{
   GP1:
	UF : 0, UT : 6,		CONFIG : 'N U T, 0, 0, 0',
	X =  86.098  mm,	Y =   -325.515  mm,	Z =   -315.922  mm,
	W =  90.000 deg,	P =   0.000 deg,	R =   90.000 deg
};
P[504]{
   GP1:
	UF : 0, UT : 6,		CONFIG : 'N U T, 0, 0, 0',
	X =  86.123  mm,	Y =   -325.558  mm,	Z =   -312.152  mm,
	W =  90.000 deg,	P =   0.000 deg,	R =   90.000 deg
};
P[505]{
   GP1:
	UF : 0, UT : 6,		CONFIG : 'N U T, 0, 0, 0',
	X =  86.157  mm,	Y =   -325.618  mm,	Z =   -311.256  mm,
	W =  90.000 deg,	P =   0.000 deg,	R =   90.000 deg
};
P[506]{
   GP1:
	UF : 0, UT : 6,		CONFIG : 'N U T, 0, 0, 0',
	X =  86.167  mm,	Y =   -325.635  mm,	Z =   -310.392  mm,
	W =  90.000 deg,	P =   0.000 deg,	R =   90.000 deg
};
P[507]{
   GP1:
	UF : 0, UT : 6,		CONFIG : 'N U T, 0, 0, 0',
	X =  86.214  mm,	Y =   -325.578  mm,	Z =   -311.016  mm,
	W =  90.000 deg,	P =   0.000 deg,	R =   90.000 deg
};
P[508]{
   GP1:
	UF : 0, UT : 6,		CONFIG : 'N U T, 0, 0, 0',
	X =  86.494  mm,	Y =   -325.121  mm,	Z =   -316.091  mm,
	W =  90.000 deg,	P =   0.000 deg,	R =   90.000 deg
};
P[509]{
   GP1:
	UF : 0, UT : 6,		CONFIG : 'N U T, 0, 0, 0',
	X =  86.985  mm,	Y =   -324.610  mm,	Z =   -324.209  mm,
	W =  90.000 deg,	P =   0.000 deg,	R =   90.000 deg
};
P[510]{
   GP1:
	UF : 0, UT : 6,		CONFIG : 'N U T, 0, 0, 0',
	X =  88.920  mm,	Y =   -323.382  mm,	Z =   -322.558  mm,
	W =  90.000 deg,	P =   0.000 deg,	R =   90.000 deg
};
P[511]{
   GP1:
	UF : 0, UT : 6,		CONFIG : 'N U T, 0, 0, 0',
	X =  89.750  mm,	Y =   -322.784  mm,	Z =   -318.920  mm,
	W =  90.000 deg,	P =   0.000 deg,	R =   90.000 deg
};
P[512]{
   GP1:
	UF : 0, UT : 6,		CONFIG : 'N U T, 0, 0, 0',
	X =  90.320  mm,	Y =   -322.347  mm,	Z =   -318.045  mm,
	W =  90.000 deg,	P =   0.000 deg,	R =   90.000 deg
};
P[513]{
   GP1:
	UF : 0, UT : 6,		CONFIG : 'N U T, 0, 0, 0',
	X =  91.620  mm,	Y =   -321.990  mm,	Z =   -325.433  mm,
	W =  90.000 deg,	P =   0.000 deg,	R =   90.000 deg
};
P[514]{
   GP1:
	UF : 0, UT : 6,		CONFIG : 'N U T, 0, 0, 0',
	X =  92.562  mm,	Y =   -321.044  mm,	Z =   -321.327  mm,
	W =  90.000 deg,	P =   0.000 deg,	R =   90.000 deg
};
P[515]{
   GP1:
	UF : 0, UT : 6,		CONFIG : 'N U T, 0, 0, 0',
	X =  95.212  mm,	Y =   -320.224  mm,	Z =   -317.240  mm,
	W =  90.000 deg,	P =   0.000 deg,	R =   90.000 deg
};
P[516]{
   GP1:
	UF : 0, UT : 6,		CONFIG : 'N U T, 0, 0, 0',
	X =  95.841  mm,	Y =   -319.679  mm,	Z =   -314.089  mm,
	W =  90.000 deg,	P =   0.000 deg,	R =   90.000 deg
};
P[517]{
   GP1:
	UF : 0, UT : 6,		CONFIG : 'N U T, 0, 0, 0',
	X =  96.867  mm,	Y =   -318.886  mm,	Z =   -325.300  mm,
	W =  90.000 deg,	P =   0.000 deg,	R =   90.000 deg
};
P[518]{
   GP1:
	UF : 0, UT : 6,		CONFIG : 'N U T, 0, 0, 0',
	X =  97.903  mm,	Y =   -318.445  mm,	Z =   -321.110  mm,
	W =  90.000 deg,	P =   0.000 deg,	R =   90.000 deg
};
P[519]{
   GP1:
	UF : 0, UT : 6,		CONFIG : 'N U T, 0, 0, 0',
	X =  99.201  mm,	Y =   -317.869  mm,	Z =   -322.286  mm,
	W =  90.000 deg,	P =   0.000 deg,	R =   90.000 deg
};
P[520]{
   GP1:
	UF : 0, UT : 6,		CONFIG : 'N U T, 0, 0, 0',
	X =  100.203  mm,	Y =   -317.120  mm,	Z =   -309.412  mm,
	W =  90.000 deg,	P =   0.000 deg,	R =   90.000 deg
};
P[521]{
   GP1:
	UF : 0, UT : 6,		CONFIG : 'N U T, 0, 0, 0',
	X =  101.057  mm,	Y =   -316.370  mm,	Z =   -318.982  mm,
	W =  90.000 deg,	P =   0.000 deg,	R =   90.000 deg
};
P[522]{
   GP1:
	UF : 0, UT : 6,		CONFIG : 'N U T, 0, 0, 0',
	X =  102.792  mm,	Y =   -315.250  mm,	Z =   -317.448  mm,
	W =  90.000 deg,	P =   0.000 deg,	R =   90.000 deg
};
P[523]{
   GP1:
	UF : 0, UT : 6,		CONFIG : 'N U T, 0, 0, 0',
	X =  103.849  mm,	Y =   -315.524  mm,	Z =   -312.779  mm,
	W =  90.000 deg,	P =   0.000 deg,	R =   90.000 deg
};
P[524]{
   GP1:
	UF : 0, UT : 6,		CONFIG : 'N U T, 0, 0, 0',
	X =  104.496  mm,	Y =   -314.697  mm,	Z =   -314.454  mm,
	W =  90.000 deg,	P =   0.000 deg,	R =   90.000 deg
};
P[525]{
   GP1:
	UF : 0, UT : 6,		CONFIG : 'N U T, 0, 0, 0',
	X =  106.266  mm,	Y =   -313.555  mm,	Z =   -324.750  mm,
	W =  90.000 deg,	P =   0.000 deg,	R =   90.000 deg
};
P[526]{
   GP1:
	UF : 0, UT : 6,		CONFIG : 'N U T, 0, 0, 0',
	X =  107.333  mm,	Y =   -313.197  mm,	Z =   -324.509  mm,
	W =  90.000 deg,	P =   0.000 deg,	R =   90.000 deg
};
P[527]{
   GP1:
	UF : 0, UT : 6,		CONFIG : 'N U T, 0, 0, 0',
	X =  108.081  mm,	Y =   -312.658  mm,	Z =   -317.276  mm,
	W =  90.000 deg,	P =   0.000 deg,	R =   90.000 deg
};
P[528]{
   GP1:
	UF : 0, UT : 6,		CONFIG : 'N U T, 0, 0, 0',
	X =  108.829  mm,	Y =   -312.410  mm,	Z =   -313.364  mm,
	W =  90.000 deg,	P =   0.000 deg,	R =   90.000 deg
};
P[529]{
   GP1:
	UF : 0, UT : 6,		CONFIG : 'N U T, 0, 0, 0',
	X =  109.721  mm,	Y =   -312.204  mm,	Z =   -320.713  mm,
	W =  90.000 deg,	P =   0.000 deg,	R =   90.000 deg
};
P[530]{
   GP1:
	UF : 0, UT : 6,		CONFIG : 'N U T, 0, 0, 0',
	X =  110.088  mm,	Y =   -311.571  mm,	Z =   -326.647  mm,
	W =  90.000 deg,	P =   0.000 deg,	R =   90.000 deg
};
P[531]{
   GP1:
	UF : 0, UT : 6,		CONFIG : 'N U T, 0, 0, 0',
	X =  110.872  mm,	Y =   -311.463  mm,	Z =   -314.253  mm,
	W =  90.000 deg,	P =   0.000 deg,	R =   90.000 deg
};
P[532]{
   GP1:
	UF : 0, UT : 6,		CONFIG : 'N U T, 0, 0, 0',
	X =  111.436  mm,	Y =   -310.855  mm,	Z =   -319.067  mm,
	W =  90.000 deg,	P =   0.000 deg,	R =   90.000 deg
};
P[533]{
   GP1:
	UF : 0, UT : 6,		CONFIG : 'N U T, 0, 0, 0',
	X =  112.623  mm,	Y =   -310.411  mm,	Z =   -313.217  mm,
	W =  90.000 deg,	P =   0.000 deg,	R =   90.000 deg
};
P[534]{
   GP1:
	UF : 0, UT : 6,		CONFIG : 'N U T, 0, 0, 0',
	X =  113.766  mm,	Y =   -309.014  mm,	Z =   -318.097  mm,
	W =  90.000 deg,	P =   0.000 deg,	R =   90.000 deg
};
P[535]{
   GP1:
	UF : 0, UT : 6,		CONFIG : 'N U T, 0, 0, 0',
	X =  114.898  mm,	Y =   -308.550  mm,	Z =   -325.675  mm,
	W =  90.000 deg,	P =   0.000 deg,	R =   90.000 deg
};
P[536]{
   GP1:
	UF : 0, UT : 6,		CONFIG : 'N U T, 0, 0, 0',
	X =  115.850  mm,	Y =   -307.790  mm,	Z =   -317.833  mm,
	W =  90.000 deg,	P =   0.000 deg,	R =   90.000 deg
};
P[537]{
   GP1:
	UF : 0, UT : 6,		CONFIG : 'N U T, 0, 0, 0',
	X =  117.282  mm,	Y =   -307.297  mm,	Z =   -313.063  mm,
	W =  90.000 deg,	P =   0.000 deg,	R =   90.000 deg
};
P[538]{
   GP1:
	UF : 0, UT : 6,		CONFIG : 'N U T, 0, 0, 0',
	X =  118.675  mm,	Y =   -306.639  mm,	Z =   -322.034  mm,
	W =  90.000 deg,	P =   0.000 deg,	R =   90.000 deg
};
P[539]{
   GP1:
	UF : 0, UT : 6,		CONFIG : 'N U T, 0, 0, 0',
	X =  119.849  mm,	Y =   -305.946  mm,	Z =   -324.753  mm,
	W =  90.000 deg,	P =   0.000 deg,	R =   90.000 deg
};
P[540]{
   GP1:
	UF : 0, UT : 6,		CONFIG : 'N U T, 0, 0, 0',
	X =  120.438  mm,	Y =   -305.193  mm,	Z =   -320.201  mm,
	W =  90.000 deg,	P =   0.000 deg,	R =   90.000 deg
};
P[541]{
   GP1:
	UF : 0, UT : 6,		CONFIG : 'N U T, 0, 0, 0',
	X =  121.594  mm,	Y =   -305.361  mm,	Z =   -322.205  mm,
	W =  90.000 deg,	P =   0.000 deg,	R =   90.000 deg
};
P[542]{
   GP1:
	UF : 0, UT : 6,		CONFIG : 'N U T, 0, 0, 0',
	X =  121.469  mm,	Y =   -304.471  mm,	Z =   -315.038  mm,
	W =  90.000 deg,	P =   0.000 deg,	R =   90.000 deg
};
P[543]{
   GP1:
	UF : 0, UT : 6,		CONFIG : 'N U T, 0, 0, 0',
	X =  122.297  mm,	Y =   -304.234  mm,	Z =   -322.268  mm,
	W =  90.000 deg,	P =   0.000 deg,	R =   90.000 deg
};
P[544]{
   GP1:
	UF : 0, UT : 6,		CONFIG : 'N U T, 0, 0, 0',
	X =  123.147  mm,	Y =   -303.956  mm,	Z =   -316.648  mm,
	W =  90.000 deg,	P =   0.000 deg,	R =   90.000 deg
};
P[545]{
   GP1:
	UF : 0, UT : 6,		CONFIG : 'N U T, 0, 0, 0',
	X =  124.669  mm,	Y =   -303.175  mm,	Z =   -323.446  mm,
	W =  90.000 deg,	P =   0.000 deg,	R =   90.000 deg
};
P[546]{
   GP1:
	UF : 0, UT : 6,		CONFIG : 'N U T, 0, 0, 0',
	X =  125.520  mm,	Y =   -302.407  mm,	Z =   -326.284  mm,
	W =  90.000 deg,	P =   0.000 deg,	R =   90.000 deg
};
P[547]{
   GP1:
	UF : 0, UT : 6,		CONFIG : 'N U T, 0, 0, 0',
	X =  126.408  mm,	Y =   -302.128  mm,	Z =   -326.859  mm,
	W =  90.000 deg,	P =   0.000 deg,	R =   90.000 deg
};
P[548]{
   GP1:
	UF : 0, UT : 6,		CONFIG : 'N U T, 0, 0, 0',
	X =  127.357  mm,	Y =   -301.256  mm,	Z =   -323.042  mm,
	W =  90.000 deg,	P =   0.000 deg,	R =   90.000 deg
};
P[549]{
   GP1:
	UF : 0, UT : 6,		CONFIG : 'N U T, 0, 0, 0',
	X =  128.042  mm,	Y =   -300.942  mm,	Z =   -312.508  mm,
	W =  90.000 deg,	P =   0.000 deg,	R =   90.000 deg
};
P[550]{
   GP1:
	UF : 0, UT : 6,		CONFIG : 'N U T, 0, 0, 0',
	X =  128.864  mm,	Y =   -300.643  mm,	Z =   -316.318  mm,
	W =  90.000 deg,	P =   0.000 deg,	R =   90.000 deg
};
P[551]{
   GP1:
	UF : 0, UT : 6,		CONFIG : 'N U T, 0, 0, 0',
	X =  129.777  mm,	Y =   -300.030  mm,	Z =   -321.759  mm,
	W =  90.000 deg,	P =   0.000 deg,	R =   90.000 deg
};
P[552]{
   GP1:
	UF : 0, UT : 6,		CONFIG : 'N U T, 0, 0, 0',
	X =  131.235  mm,	Y =   -299.251  mm,	Z =   -313.251  mm,
	W =  90.000 deg,	P =   0.000 deg,	R =   90.000 deg
};
P[553]{
   GP1:
	UF : 0, UT : 6,		CONFIG : 'N U T, 0, 0, 0',
	X =  132.512  mm,	Y =   -298.660  mm,	Z =   -316.744  mm,
	W =  90.000 deg,	P =   0.000 deg,	R =   90.000 deg
};
P[554]{
   GP1:
	UF : 0, UT : 6,		CONFIG : 'N U T, 0, 0, 0',
	X =  133.263  mm,	Y =   -298.142  mm,	Z =   -318.775  mm,
	W =  90.000 deg,	P =   0.000 deg,	R =   90.000 deg
};
P[555]{
   GP1:
	UF : 0, UT : 6,		CONFIG : 'N U T, 0, 0, 0',
	X =  134.098  mm,	Y =   -297.446  mm,	Z =   -309.771  mm,
	W =  90.000 deg,	P =   0.000 deg,	R =   90.000 deg
};
P[556]{
   GP1:
	UF : 0, UT : 6,		CONFIG : 'N U T, 0, 0, 0',
	X =  135.654  mm,	Y =   -296.665  mm,	Z =   -310.491  mm,
	W =  90.000 deg,	P =   0.000 deg,	R =   90.000 deg
};
P[557]{
   GP1:
	UF : 0, UT : 6,		CONFIG : 'N U T, 0, 0, 0',
	X =  136.845  mm,	Y =   -296.005  mm,	Z =   -313.044  mm,
	W =  90.000 deg,	P =   0.000 deg,	R =   90.000 deg
};
P[558]{
   GP1:
	UF : 0, UT : 6,		CONFIG : 'N U T, 0, 0, 0',
	X =  137.163  mm,	Y =   -295.332  mm,	Z =   -318.530  mm,
	W =  90.000 deg,	P =   0.000 deg,	R =   90.000 deg
};
P[559]{
   GP1:
	UF : 0, UT : 6,		CONFIG : 'N U T, 0, 0, 0',
	X =  137.829  mm,	Y =   -295.610  mm,	Z =   -320.695  mm,
	W =  90.000 deg,	P =   0.000 deg,	R =   90.000 deg
};
P[560]{
   GP1:
	UF : 0, UT : 6,		CONFIG : 'N U T, 0, 0, 0',
	X =  138.613  mm,	Y =   -295.079  mm,	Z =   -325.647  mm,
	W =  90.000 deg,	P =   0.000 deg,	R =   90.000 deg
};
P[561]{
   GP1:
	UF : 0, UT : 6,		CONFIG : 'N U T, 0, 0, 0',
	X =  139.220  mm,	Y =   -294.755  mm,	Z =   -324.283  mm,
	W =  90.000 deg,	P =   0.000 deg,	R =   90.000 deg
};
P[562]{
   GP1:
	UF : 0, UT : 6,		CONFIG : 'N U T, 0, 0, 0',
	X =  140.022  mm,	Y =   -294.393  mm,	Z =   -315.223  mm,
	W =  90.000 deg,	P =   0.000 deg,	R =   90.000 deg
};
P[563]{
   GP1:
	UF : 0, UT : 6,		CONFIG : 'N U T, 0, 0, 0',
	X =  140.974  mm,	Y =   -293.815  mm,	Z =   -325.692  mm,
	W =  90.000 deg,	P =   0.000 deg,	R =   90.000 deg
};
P[564]{
   GP1:
	UF : 0, UT : 6,		CONFIG : 'N U T, 0, 0, 0',
	X =  141.410  mm,	Y =   -293.340  mm,	Z =   -310.077  mm,
	W =  90.000 deg,	P =   0.000 deg,	R =   90.000 deg
};
P[565]{
   GP1:
	UF : 0, UT : 6,		CONFIG : 'N U T, 0, 0, 0',
	X =  142.062  mm,	Y =   -293.139  mm,	Z =   -324.115  mm,
	W =  90.000 deg,	P =   0.000 deg,	R =   90.000 deg
};
P[566]{
   GP1:
	UF : 0, UT : 6,		CONFIG : 'N U T, 0, 0, 0',
	X =  142.377  mm,	Y =   -292.346  mm,	Z =   -317.639  mm,
	W =  90.000 deg,	P =   0.000 deg,	R =   90.000 deg
};
P[567]{
   GP1:
	UF : 0, UT : 6,		CONFIG : 'N U T, 0, 0, 0',
	X =  143.254  mm,	Y =   -292.409  mm,	Z =   -326.401  mm,
	W =  90.000 deg,	P =   0.000 deg,	R =   90.000 deg
};
P[568]{
   GP1:
	UF : 0, UT : 6,		CONFIG : 'N U T, 0, 0, 0',
	X =  143.586  mm,	Y =   -291.820  mm,	Z =   -322.320  mm,
	W =  90.000 deg,	P =   0.000 deg,	R =   90.000 deg
};
P[569]{
   GP1:
	UF : 0, UT : 6,		CONFIG : 'N U T, 0, 0, 0',
	X =  144.240  mm,	Y =   -292.171  mm,	Z =   -313.017  mm,
	W =  90.000 deg,	P =   0.000 deg,	R =   90.000 deg
};
P[570]{
   GP1:
	UF : 0, UT : 6,		CONFIG : 'N U T, 0, 0, 0',
	X =  144.266  mm,	Y =   -291.492  mm,	Z =   -322.214  mm,
	W =  90.000 deg,	P =   0.000 deg,	R =   90.000 deg
};
P[571]{
   GP1:
	UF : 0, UT : 6,		CONFIG : 'N U T, 0, 0, 0',
	X =  144.841  mm,	Y =   -291.324  mm,	Z =   -322.837  mm,
	W =  90.000 deg,	P =   0.000 deg,	R =   90.000 deg
};
P[572]{
   GP1:
	UF : 0, UT : 6,		CONFIG : 'N U T, 0, 0, 0',
	X =  145.293  mm,	Y =   -290.993  mm,	Z =   -325.863  mm,
	W =  90.000 deg,	P =   0.000 deg,	R =   90.000 deg
};
P[573]{
   GP1:
	UF : 0, UT : 6,		CONFIG : 'N U T, 0, 0, 0',
	X =  145.741  mm,	Y =   -290.598  mm,	Z =   -318.149  mm,
	W =  90.000 deg,	P =   0.000 deg,	R =   90.000 deg
};
P[574]{
   GP1:
	UF : 0, UT : 6,		CONFIG : 'N U T, 0, 0, 0',
	X =  146.635  mm,	Y =   -290.424  mm,	Z =   -319.626  mm,
	W =  90.000 deg,	P =   0.000 deg,	R =   90.000 deg
};
P[575]{
   GP1:
	UF : 0, UT : 6,		CONFIG : 'N U T, 0, 0, 0',
	X =  147.107  mm,	Y =   -289.989  mm,	Z =   -323.108  mm,
	W =  90.000 deg,	P =   0.000 deg,	R =   90.000 deg
};
P[576]{
   GP1:
	UF : 0, UT : 6,		CONFIG : 'N U T, 0, 0, 0',
	X =  147.690  mm,	Y =   -289.654  mm,	Z =   -323.595  mm,
	W =  90.000 deg,	P =   0.000 deg,	R =   90.000 deg
};
P[577]{
   GP1:
	UF : 0, UT : 6,		CONFIG : 'N U T, 0, 0, 0',
	X =  148.921  mm,	Y =   -288.857  mm,	Z =   -323.528  mm,
	W =  90.000 deg,	P =   0.000 deg,	R =   90.000 deg
};
P[578]{
   GP1:
	UF : 0, UT : 6,		CONFIG : 'N U T, 0, 0, 0',
	X =  149.779  mm,	Y =   -287.977  mm,	Z =   -321.469  mm,
	W =  90.000 deg,	P =   0.000 deg,	R =   90.000 deg
};
P[579]{
   GP1:
	UF : 0, UT : 6,		CONFIG : 'N U T, 0, 0, 0',
	X =  150.428  mm,	Y =   -288.348  mm,	Z =   -317.901  mm,
	W =  90.000 deg,	P =   0.000 deg,	R =   90.000 deg
};
P[580]{
   GP1:
	UF : 0, UT : 6,		CONFIG : 'N U T, 0, 0, 0',
	X =  151.915  mm,	Y =   -287.314  mm,	Z =   -313.395  mm,
	W =  90.000 deg,	P =   0.000 deg,	R =   90.000 deg
};
P[581]{
   GP1:
	UF : 0, UT : 6,		CONFIG : 'N U T, 0, 0, 0',
	X =  152.968  mm,	Y =   -286.678  mm,	Z =   -312.273  mm,
	W =  90.000 deg,	P =   0.000 deg,	R =   90.000 deg
};
P[582]{
   GP1:
	UF : 0, UT : 6,		CONFIG : 'N U T, 0, 0, 0',
	X =  154.288  mm,	Y =   -286.383  mm,	Z =   -312.275  mm,
	W =  90.000 deg,	P =   0.000 deg,	R =   90.000 deg
};
P[583]{
   GP1:
	UF : 0, UT : 6,		CONFIG : 'N U T, 0, 0, 0',
	X =  154.792  mm,	Y =   -285.704  mm,	Z =   -317.134  mm,
	W =  90.000 deg,	P =   0.000 deg,	R =   90.000 deg
};
P[584]{
   GP1:
	UF : 0, UT : 6,		CONFIG : 'N U T, 0, 0, 0',
	X =  155.667  mm,	Y =   -284.866  mm,	Z =   -320.279  mm,
	W =  90.000 deg,	P =   0.000 deg,	R =   90.000 deg
};
P[585]{
   GP1:
	UF : 0, UT : 6,		CONFIG : 'N U T, 0, 0, 0',
	X =  157.646  mm,	Y =   -284.105  mm,	Z =   -326.253  mm,
	W =  90.000 deg,	P =   0.000 deg,	R =   90.000 deg
};
P[586]{
   GP1:
	UF : 0, UT : 6,		CONFIG : 'N U T, 0, 0, 0',
	X =  159.575  mm,	Y =   -282.853  mm,	Z =   -311.263  mm,
	W =  90.000 deg,	P =   0.000 deg,	R =   90.000 deg
};
P[587]{
   GP1:
	UF : 0, UT : 6,		CONFIG : 'N U T, 0, 0, 0',
	X =  160.644  mm,	Y =   -282.252  mm,	Z =   -311.741  mm,
	W =  90.000 deg,	P =   0.000 deg,	R =   90.000 deg
};
P[588]{
   GP1:
	UF : 0, UT : 6,		CONFIG : 'N U T, 0, 0, 0',
	X =  161.711  mm,	Y =   -281.676  mm,	Z =   -315.979  mm,
	W =  90.000 deg,	P =   0.000 deg,	R =   90.000 deg
};
P[589]{
   GP1:
	UF : 0, UT : 6,		CONFIG : 'N U T, 0, 0, 0',
	X =  162.599  mm,	Y =   -281.111  mm,	Z =   -311.113  mm,
	W =  90.000 deg,	P =   0.000 deg,	R =   90.000 deg
};
P[590]{
   GP1:
	UF : 0, UT : 6,		CONFIG : 'N U T, 0, 0, 0',
	X =  163.479  mm,	Y =   -280.842  mm,	Z =   -316.778  mm,
	W =  90.000 deg,	P =   0.000 deg,	R =   90.000 deg
};
P[591]{
   GP1:
	UF : 0, UT : 6,		CONFIG : 'N U T, 0, 0, 0',
	X =  164.307  mm,	Y =   -279.856  mm,	Z =   -318.226  mm,
	W =  90.000 deg,	P =   0.000 deg,	R =   90.000 deg
};
P[592]{
   GP1:
	UF : 0, UT : 6,		CONFIG : 'N U T, 0, 0, 0',
	X =  165.085  mm,	Y =   -279.892  mm,	Z =   -316.393  mm,
	W =  90.000 deg,	P =   0.000 deg,	R =   90.000 deg
};
P[593]{
   GP1:
	UF : 0, UT : 6,		CONFIG : 'N U T, 0, 0, 0',
	X =  166.672  mm,	Y =   -278.996  mm,	Z =   -317.224  mm,
	W =  90.000 deg,	P =   0.000 deg,	R =   90.000 deg
};
P[594]{
   GP1:
	UF : 0, UT : 6,		CONFIG : 'N U T, 0, 0, 0',
	X =  167.548  mm,	Y =   -278.838  mm,	Z =   -321.458  mm,
	W =  90.000 deg,	P =   0.000 deg,	R =   90.000 deg
};
P[595]{
   GP1:
	UF : 0, UT : 6,		CONFIG : 'N U T, 0, 0, 0',
	X =  167.768  mm,	Y =   -277.846  mm,	Z =   -319.202  mm,
	W =  90.000 deg,	P =   0.000 deg,	R =   90.000 deg
};
P[596]{
   GP1:
	UF : 0, UT : 6,		CONFIG : 'N U T, 0, 0, 0',
	X =  168.133  mm,	Y =   -277.606  mm,	Z =   -322.914  mm,
	W =  90.000 deg,	P =   0.000 deg,	R =   90.000 deg
};
P[597]{
   GP1:
	UF : 0, UT : 6,		CONFIG : 'N U T, 0, 0, 0',
	X =  168.220  mm,	Y =   -277.756  mm,	Z =   -323.815  mm,
	W =  90.000 deg,	P =   0.000 deg,	R =   90.000 deg
};
P[598]{
   GP1:
	UF : 0, UT : 6,		CONFIG : 'N U T, 0, 0, 0',
	X =  168.239  mm,	Y =   -277.789  mm,	Z =   -323.144  mm,
	W =  90.000 deg,	P =   0.000 deg,	R =   90.000 deg
};
P[599]{
   GP1:
	UF : 0, UT : 6,		CONFIG : 'N U T, 0, 0, 0',
	X =  168.263  mm,	Y =   -277.831  mm,	Z =   -310.370  mm,
	W =  90.000 deg,	P =   0.000 deg,	R =   90.000 deg
};
P[600]{
   GP1:
	UF : 0, UT : 6,		CONFIG : 'N U T, 0, 0, 0',
	X =  168.318  mm,	Y =   -277.925  mm,	Z =   -314.183  mm,
	W =  90.000 deg,	P =   0.000 deg,	R =   90.000 deg
};
P[601]{
   GP1:
	UF : 0, UT : 6,		CONFIG : 'N U T, 0, 0, 0',
	X =  168.319  mm,	Y =   -277.927  mm,	Z =   -324.545  mm,
	W =  90.000 deg,	P =   0.000 deg,	R =   90.000 deg
};
P[602]{
   GP1:
	UF : 0, UT : 6,		CONFIG : 'N U T, 0, 0, 0',
	X =  168.354  mm,	Y =   -277.987  mm,	Z =   -320.017  mm,
	W =  90.000 deg,	P =   0.000 deg,	R =   90.000 deg
};
P[603]{
   GP1:
	UF : 0, UT : 6,		CONFIG : 'N U T, 0, 0, 0',
	X =  168.436  mm,	Y =   -278.129  mm,	Z =   -311.294  mm,
	W =  90.000 deg,	P =   0.000 deg,	R =   90.000 deg
};
P[604]{
   GP1:
	UF : 0, UT : 6,		CONFIG : 'N U T, 0, 0, 0',
	X =  168.442  mm,	Y =   -278.140  mm,	Z =   -310.005  mm,
	W =  90.000 deg,	P =   0.000 deg,	R =   90.000 deg
};
P[605]{
   GP1:
	UF : 0, UT : 6,		CONFIG : 'N U T, 0, 0, 0',
	X =  168.496  mm,	Y =   -278.096  mm,	Z =   -310.978  mm,
	W =  90.000 deg,	P =   0.000 deg,	R =   90.000 deg
};
P[606]{
   GP1:
	UF : 0, UT : 6,		CONFIG : 'N U T, 0, 0, 0',
	X =  168.788  mm,	Y =   -277.869  mm,	Z =   -312.243  mm,
	W =  90.000 deg,	P =   0.000 deg,	R =   90.000 deg
};
P[607]{
   GP1:
	UF : 0, UT : 6,		CONFIG : 'N U T, 0, 0, 0',
	X =  169.560  mm,	Y =   -277.107  mm,	Z =   -312.889  mm,
	W =  90.000 deg,	P =   0.000 deg,	R =   90.000 deg
};
P[608]{
   GP1:
	UF : 0, UT : 6,		CONFIG : 'N U T, 0, 0, 0',
	X =  171.085  mm,	Y =   -276.457  mm,	Z =   -315.082  mm,
	W =  90.000 deg,	P =   0.000 deg,	R =   90.000 deg
};
P[609]{
   GP1:
	UF : 0, UT : 6,		CONFIG : 'N U T, 0, 0, 0',
	X =  172.073  mm,	Y =   -275.915  mm,	Z =   -312.828  mm,
	W =  90.000 deg,	P =   0.000 deg,	R =   90.000 deg
};
P[610]{
   GP1:
	UF : 0, UT : 6,		CONFIG : 'N U T, 0, 0, 0',
	X =  173.044  mm,	Y =   -275.134  mm,	Z =   -316.051  mm,
	W =  90.000 deg,	P =   0.000 deg,	R =   90.000 deg
};
P[611]{
   GP1:
	UF : 0, UT : 6,		CONFIG : 'N U T, 0, 0, 0',
	X =  173.903  mm,	Y =   -274.784  mm,	Z =   -319.182  mm,
	W =  90.000 deg,	P =   0.000 deg,	R =   90.000 deg
};
P[612]{
   GP1:
	UF : 0, UT : 6,		CONFIG : 'N U T, 0, 0, 0',
	X =  175.702  mm,	Y =   -273.615  mm,	Z =   -318.023  mm,
	W =  90.000 deg,	P =   0.000 deg,	R =   90.000 deg
};
P[613]{
   GP1:
	UF : 0, UT : 6,		CONFIG : 'N U T, 0, 0, 0',
	X =  176.601  mm,	Y =   -273.160  mm,	Z =   -327.664  mm,
	W =  90.000 deg,	P =   0.000 deg,	R =   90.000 deg
};
P[614]{
   GP1:
	UF : 0, UT : 6,		CONFIG : 'N U T, 0, 0, 0',
	X =  177.170  mm,	Y =   -272.724  mm,	Z =   -313.636  mm,
	W =  90.000 deg,	P =   0.000 deg,	R =   90.000 deg
};
P[615]{
   GP1:
	UF : 0, UT : 6,		CONFIG : 'N U T, 0, 0, 0',
	X =  177.901  mm,	Y =   -272.550  mm,	Z =   -312.614  mm,
	W =  90.000 deg,	P =   0.000 deg,	R =   90.000 deg
};
P[616]{
   GP1:
	UF : 0, UT : 6,		CONFIG : 'N U T, 0, 0, 0',
	X =  178.706  mm,	Y =   -272.298  mm,	Z =   -315.021  mm,
	W =  90.000 deg,	P =   0.000 deg,	R =   90.000 deg
};
P[617]{
   GP1:
	UF : 0, UT : 6,		CONFIG : 'N U T, 0, 0, 0',
	X =  179.439  mm,	Y =   -271.091  mm,	Z =   -322.684  mm,
	W =  90.000 deg,	P =   0.000 deg,	R =   90.000 deg
};
P[618]{
   GP1:
	UF : 0, UT : 6,		CONFIG : 'N U T, 0, 0, 0',
	X =  180.542  mm,	Y =   -270.834  mm,	Z =   -317.403  mm,
	W =  90.000 deg,	P =   0.000 deg,	R =   90.000 deg
};
P[619]{
   GP1:
	UF : 0, UT : 6,		CONFIG : 'N U T, 0, 0, 0',
	X =  182.084  mm,	Y =   -269.818  mm,	Z =   -322.450  mm,
	W =  90.000 deg,	P =   0.000 deg,	R =   90.000 deg
};
P[620]{
   GP1:
	UF : 0, UT : 6,		CONFIG : 'N U T, 0, 0, 0',
	X =  182.860  mm,	Y =   -269.670  mm,	Z =   -313.845  mm,
	W =  90.000 deg,	P =   0.000 deg,	R =   90.000 deg
};
P[621]{
   GP1:
	UF : 0, UT : 6,		CONFIG : 'N U T, 0, 0, 0',
	X =  183.111  mm,	Y =   -268.895  mm,	Z =   -317.601  mm,
	W =  90.000 deg,	P =   0.000 deg,	R =   90.000 deg
};
P[622]{
   GP1:
	UF : 0, UT : 6,		CONFIG : 'N U T, 0, 0, 0',
	X =  183.815  mm,	Y =   -268.638  mm,	Z =   -323.814  mm,
	W =  90.000 deg,	P =   0.000 deg,	R =   90.000 deg
};
P[623]{
   GP1:
	UF : 0, UT : 6,		CONFIG : 'N U T, 0, 0, 0',
	X =  185.092  mm,	Y =   -268.119  mm,	Z =   -310.256  mm,
	W =  90.000 deg,	P =   0.000 deg,	R =   90.000 deg
};
P[624]{
   GP1:
	UF : 0, UT : 6,		CONFIG : 'N U T, 0, 0, 0',
	X =  185.514  mm,	Y =   -267.522  mm,	Z =   -322.350  mm,
	W =  90.000 deg,	P =   0.000 deg,	R =   90.000 deg
};
P[625]{
   GP1:
	UF : 0, UT : 6,		CONFIG : 'N U T, 0, 0, 0',
	X =  186.431  mm,	Y =   -266.968  mm,	Z =   -317.029  mm,
	W =  90.000 deg,	P =   0.000 deg,	R =   90.000 deg
};
P[626]{
   GP1:
	UF : 0, UT : 6,		CONFIG : 'N U T, 0, 0, 0',
	X =  187.307  mm,	Y =   -267.094  mm,	Z =   -314.112  mm,
	W =  90.000 deg,	P =   0.000 deg,	R =   90.000 deg
};
P[627]{
   GP1:
	UF : 0, UT : 6,		CONFIG : 'N U T, 0, 0, 0',
	X =  188.100  mm,	Y =   -266.407  mm,	Z =   -313.817  mm,
	W =  90.000 deg,	P =   0.000 deg,	R =   90.000 deg
};
P[628]{
   GP1:
	UF : 0, UT : 6,		CONFIG : 'N U T, 0, 0, 0',
	X =  188.818  mm,	Y =   -266.083  mm,	Z =   -319.793  mm,
	W =  90.000 deg,	P =   0.000 deg,	R =   90.000 deg
};
P[629]{
   GP1:
	UF : 0, UT : 6,		CONFIG : 'N U T, 0, 0, 0',
	X =  190.780  mm,	Y =   -264.829  mm,	Z =   -310.659  mm,
	W =  90.000 deg,	P =   0.000 deg,	R =   90.000 deg
};
P[630]{
   GP1:
	UF : 0, UT : 6,		CONFIG : 'N U T, 0, 0, 0',
	X =  191.558  mm,	Y =   -264.692  mm,	Z =   -311.762  mm,
	W =  90.000 deg,	P =   0.000 deg,	R =   90.000 deg
};
P[631]{
   GP1:
	UF : 0, UT : 6,		CONFIG : 'N U T, 0, 0, 0',
	X =  192.158  mm,	Y =   -263.944  mm,	Z =   -325.443  mm,
	W =  90.000 deg,	P =   0.000 deg,	R =   90.000 deg
};
P[632]{
   GP1:
	UF : 0, UT : 6,		CONFIG : 'N U T, 0, 0, 0',
	X =  192.852  mm,	Y =   -263.176  mm,	Z =   -320.095  mm,
	W =  90.000 deg,	P =   0.000 deg,	R =   90.000 deg
};
P[633]{
   GP1:
	UF : 0, UT : 6,		CONFIG : 'N U T, 0, 0, 0',
	X =  193.667  mm,	Y =   -263.550  mm,	Z =   -311.502  mm,
	W =  90.000 deg,	P =   0.000 deg,	R =   90.000 deg
};
P[634]{
   GP1:
	UF : 0, UT : 6,		CONFIG : 'N U T, 0, 0, 0',
	X =  194.797  mm,	Y =   -262.416  mm,	Z =   -327.027  mm,
	W =  90.000 deg,	P =   0.000 deg,	R =   90.000 deg
};
P[635]{
   GP1:
	UF : 0, UT : 6,		CONFIG : 'N U T, 0, 0, 0',
	X =  195.757  mm,	Y =   -262.112  mm,	Z =   -324.914  mm,
	W =  90.000 deg,	P =   0.000 deg,	R =   90.000 deg
};
P[636]{
   GP1:
	UF : 0, UT : 6,		CONFIG : 'N U T, 0, 0, 0',
	X =  196.522  mm,	Y =   -261.290  mm,	Z =   -319.894  mm,
	W =  90.000 deg,	P =   0.000 deg,	R =   90.000 deg
};
P[637]{
   GP1:
	UF : 0, UT : 6,		CONFIG : 'N U T, 0, 0, 0',
	X =  197.339  mm,	Y =   -260.992  mm,	Z =   -324.127  mm,
	W =  90.000 deg,	P =   0.000 deg,	R =   90.000 deg
};
P[638]{
   GP1:
	UF : 0, UT : 6,		CONFIG : 'N U T, 0, 0, 0',
	X =  198.170  mm,	Y =   -260.444  mm,	Z =   -323.500  mm,
	W =  90.000 deg,	P =   0.000 deg,	R =   90.000 deg
};
P[639]{
   GP1:
	UF : 0, UT : 6,		CONFIG : 'N U T, 0, 0, 0',
	X =  198.880  mm,	Y =   -260.662  mm,	Z =   -316.130  mm,
	W =  90.000 deg,	P =   0.000 deg,	R =   90.000 deg
};
P[640]{
   GP1:
	UF : 0, UT : 6,		CONFIG : 'N U T, 0, 0, 0',
	X =  200.270  mm,	Y =   -259.376  mm,	Z =   -314.213  mm,
	W =  90.000 deg,	P =   0.000 deg,	R =   90.000 deg
};
P[641]{
   GP1:
	UF : 0, UT : 6,		CONFIG : 'N U T, 0, 0, 0',
	X =  201.049  mm,	Y =   -259.104  mm,	Z =   -320.487  mm,
	W =  90.000 deg,	P =   0.000 deg,	R =   90.000 deg
};
P[642]{
   GP1:
	UF : 0, UT : 6,		CONFIG : 'N U T, 0, 0, 0',
	X =  201.750  mm,	Y =   -258.244  mm,	Z =   -319.632  mm,
	W =  90.000 deg,	P =   0.000 deg,	R =   90.000 deg
};
P[643]{
   GP1:
	UF : 0, UT : 6,		CONFIG : 'N U T, 0, 0, 0',
	X =  202.799  mm,	Y =   -258.082  mm,	Z =   -316.486  mm,
	W =  90.000 deg,	P =   0.000 deg,	R =   90.000 deg
};
P[644]{
   GP1:
	UF : 0, UT : 6,		CONFIG : 'N U T, 0, 0, 0',
	X =  203.614  mm,	Y =   -257.189  mm,	Z =   -320.100  mm,
	W =  90.000 deg,	P =   0.000 deg,	R =   90.000 deg
};
P[645]{
   GP1:
	UF : 0, UT : 6,		CONFIG : 'N U T, 0, 0, 0',
	X =  204.590  mm,	Y =   -257.191  mm,	Z =   -312.089  mm,
	W =  90.000 deg,	P =   0.000 deg,	R =   90.000 deg
};
P[646]{
   GP1:
	UF : 0, UT : 6,		CONFIG : 'N U T, 0, 0, 0',
	X =  205.331  mm,	Y =   -256.383  mm,	Z =   -323.744  mm,
	W =  90.000 deg,	P =   0.000 deg,	R =   90.000 deg
};
P[647]{
   GP1:
	UF : 0, UT : 6,		CONFIG : 'N U T, 0, 0, 0',
	X =  206.426  mm,	Y =   -256.024  mm,	Z =   -316.134  mm,
	W =  90.000 deg,	P =   0.000 deg,	R =   90.000 deg
};
P[648]{
   GP1:
	UF : 0, UT : 6,		CONFIG : 'N U T, 0, 0, 0',
	X =  206.877  mm,	Y =   -255.089  mm,	Z =   -319.457  mm,
	W =  90.000 deg,	P =   0.000 deg,	R =   90.000 deg
};
P[649]{
   GP1:
	UF : 0, UT : 6,		CONFIG : 'N U T, 0, 0, 0',
	X =  207.842  mm,	Y =   -255.172  mm,	Z =   -320.653  mm,
	W =  90.000 deg,	P =   0.000 deg,	R =   90.000 deg
};
P[650]{
   GP1:
	UF : 0, UT : 6,		CONFIG : 'N U T, 0, 0, 0',
	X =  208.767  mm,	Y =   -254.971  mm,	Z =   -319.346  mm,
	W =  90.000 deg,	P =   0.000 deg,	R =   90.000 deg
};
P[651]{
   GP1:
	UF : 0, UT : 6,		CONFIG : 'N U T, 0, 0, 0',
	X =  209.425  mm,	Y =   -253.803  mm,	Z =   -320.326  mm,
	W =  90.000 deg,	P =   0.000 deg,	R =   90.000 deg
};
P[652]{
   GP1:
	UF : 0, UT : 6,		CONFIG : 'N U T, 0, 0, 0',
	X =  210.091  mm,	Y =   -253.377  mm,	Z =   -317.406  mm,
	W =  90.000 deg,	P =   0.000 deg,	R =   90.000 deg
};
P[653]{
   GP1:
	UF : 0, UT : 6,		CONFIG : 'N U T, 0, 0, 0',
	X =  211.038  mm,	Y =   -253.551  mm,	Z =   -310.168  mm,
	W =  90.000 deg,	P =   0.000 deg,	R =   90.000 deg
};
P[654]{
   GP1:
	UF : 0, UT : 6,		CONFIG : 'N U T, 0, 0, 0',
	X =  211.645  mm,	Y =   -252.981  mm,	Z =   -321.002  mm,
	W =  90.000 deg,	P =   0.000 deg,	R =   90.000 deg
};
P[655]{
   GP1:
	UF : 0, UT : 6,		CONFIG : 'N U T, 0, 0, 0',
	X =  212.325  mm,	Y =   -252.476  mm,	Z =   -318.082  mm,
	W =  90.000 deg,	P =   0.000 deg,	R =   90.000 deg
};
P[656]{
   GP1:
	UF : 0, UT : 6,		CONFIG : 'N U T, 0, 0, 0',
	X =  213.630  mm,	Y =   -252.165  mm,	Z =   -319.952  mm,
	W =  90.000 deg,	P =   0.000 deg,	R =   90.000 deg
};
P[657]{
   GP1:
	UF : 0, UT : 6,		CONFIG : 'N U T, 0, 0, 0',
	X =  214.747  mm,	Y =   -251.045  mm,	Z =   -314.637  mm,
	W =  90.000 deg,	P =   0.000 deg,	R =   90.000 deg
};
P[658]{
   GP1:
	UF : 0, UT : 6,		CONFIG : 'N U T, 0, 0, 0',
	X =  215.603  mm,	Y =   -250.395  mm,	Z =   -313.798  mm,
	W =  90.000 deg,	P =   0.000 deg,	R =   90.000 deg
};
P[659]{
   GP1:
	UF : 0, UT : 6,		CONFIG : 'N U T, 0, 0, 0',
	X =  216.824  mm,	Y =   -250.165  mm,	Z =   -310.867  mm,
	W =  90.000 deg,	P =   0.000 deg,	R =   90.000 deg
};
P[660]{
   GP1:
	UF : 0, UT : 6,		CONFIG : 'N U T, 0, 0, 0',
	X =  217.504  mm,	Y =   -249.461  mm,	Z =   -315.643  mm,
	W =  90.000 deg,	P =   0.000 deg,	R =   90.000 deg
};
P[661]{
   GP1:
	UF : 0, UT : 6,		CONFIG : 'N U T, 0, 0, 0',
	X =  218.217  mm,	Y =   -249.152  mm,	Z =   -322.741  mm,
	W =  90.000 deg,	P =   0.000 deg,	R =   90.000 deg
};
P[662]{
   GP1:
	UF : 0, UT : 6,		CONFIG : 'N U T, 0, 0, 0',
	X =  218.875  mm,	Y =   -248.686  mm,	Z =   -317.246  mm,
	W =  90.000 deg,	P =   0.000 deg,	R =   90.000 deg
};
P[663]{
   GP1:
	UF : 0, UT : 6,		CONFIG : 'N U T, 0, 0, 0',
	X =  219.794  mm,	Y =   -248.124  mm,	Z =   -314.822  mm,
	W =  90.000 deg,	P =   0.000 deg,	R =   90.000 deg
};
P[664]{
   GP1:
	UF : 0, UT : 6,		CONFIG : 'N U T, 0, 0, 0',
	X =  219.960  mm,	Y =   -247.462  mm,	Z =   -320.236  mm,
	W =  90.000 deg,	P =   0.000 deg,	R =   90.000 deg
};
P[665]{
   GP1:
	UF : 0, UT : 6,		CONFIG : 'N U T, 0, 0, 0',
	X =  220.608  mm,	Y =   -247.398  mm,	Z =   -323.551  mm,
	W =  90.000 deg,	P =   0.000 deg,	R =   90.000 deg
};
P[666]{
   GP1:
	UF : 0, UT : 6,		CONFIG : 'N U T, 0, 0, 0',
	X =  221.521  mm,	Y =   -247.037  mm,	Z =   -322.063  mm,
	W =  90.000 deg,	P =   0.000 deg,	R =   90.000 deg
};
P[667]{
   GP1:
	UF : 0, UT : 6,		CONFIG : 'N U T, 0, 0, 0',
	X =  222.694  mm,	Y =   -246.413  mm,	Z =   -311.643  mm,
	W =  90.000 deg,	P =   0.000 deg,	R =   90.000 deg
};
P[668]{
   GP1:
	UF : 0, UT : 6,		CONFIG : 'N U T, 0, 0, 0',
	X =  223.297  mm,	Y =   -245.652  mm,	Z =   -316.933  mm,
	W =  90.000 deg,	P =   0.000 deg,	R =   90.000 deg
};
P[669]{
   GP1:
	UF : 0, UT : 6,		CONFIG : 'N U T, 0, 0, 0',
	X =  224.141  mm,	Y =   -245.612  mm,	Z =   -315.049  mm,
	W =  90.000 deg,	P =   0.000 deg,	R =   90.000 deg
};
P[670]{
   GP1:
	UF : 0, UT : 6,		CONFIG : 'N U T, 0, 0, 0',
	X =  224.824  mm,	Y =   -245.106  mm,	Z =   -326.719  mm,
	W =  90.000 deg,	P =   0.000 deg,	R =   90.000 deg
};
P[671]{
   GP1:
	UF : 0, UT : 6,		CONFIG : 'N U T, 0, 0, 0',
	X =  225.287  mm,	Y =   -244.659  mm,	Z =   -321.024  mm,
	W =  90.000 deg,	P =   0.000 deg,	R =   90.000 deg
};
P[672]{
   GP1:
	UF : 0, UT : 6,		CONFIG : 'N U T, 0, 0, 0',
	X =  225.974  mm,	Y =   -244.597  mm,	Z =   -318.674  mm,
	W =  90.000 deg,	P =   0.000 deg,	R =   90.000 deg
};
P[673]{
   GP1:
	UF : 0, UT : 6,		CONFIG : 'N U T, 0, 0, 0',
	X =  226.472  mm,	Y =   -243.991  mm,	Z =   -319.118  mm,
	W =  90.000 deg,	P =   0.000 deg,	R =   90.000 deg
};
P[674]{
   GP1:
	UF : 0, UT : 6,		CONFIG : 'N U T, 0, 0, 0',
	X =  227.965  mm,	Y =   -243.186  mm,	Z =   -324.774  mm,
	W =  90.000 deg,	P =   0.000 deg,	R =   90.000 deg
};
P[675]{
   GP1:
	UF : 0, UT : 6,		CONFIG : 'N U T, 0, 0, 0',
	X =  228.495  mm,	Y =   -243.461  mm,	Z =   -309.966  mm,
	W =  90.000 deg,	P =   0.000 deg,	R =   90.000 deg
};
P[676]{
   GP1:
	UF : 0, UT : 6,		CONFIG : 'N U T, 0, 0, 0',
	X =  228.729  mm,	Y =   -243.128  mm,	Z =   -318.283  mm,
	W =  90.000 deg,	P =   0.000 deg,	R =   90.000 deg
};
P[677]{
   GP1:
	UF : 0, UT : 6,		CONFIG : 'N U T, 0, 0, 0',
	X =  228.944  mm,	Y =   -243.015  mm,	Z =   -319.025  mm,
	W =  90.000 deg,	P =   0.000 deg,	R =   90.000 deg
};
P[678]{
   GP1:
	UF : 0, UT : 6,		CONFIG : 'N U T, 0, 0, 0',
	X =  229.449  mm,	Y =   -242.580  mm,	Z =   -315.010  mm,
	W =  90.000 deg,	P =   0.000 deg,	R =   90.000 deg
};
P[679]{
   GP1:
	UF : 0, UT : 6,		CONFIG : 'N U T, 0, 0, 0',
	X =  230.095  mm,	Y =   -241.757  mm,	Z =   -316.370  mm,
	W =  90.000 deg,	P =   0.000 deg,	R =   90.000 deg
};
P[680]{
   GP1:
	UF : 0, UT : 6,		CONFIG : 'N U T, 0, 0, 0',
	X =  231.016  mm,	Y =   -241.151  mm,	Z =   -319.201  mm,
	W =  90.000 deg,	P =   0.000 deg,	R =   90.000 deg
};
P[681]{
   GP1:
	UF : 0, UT : 6,		CONFIG : 'N U T, 0, 0, 0',
	X =  231.921  mm,	Y =   -241.016  mm,	Z =   -321.979  mm,
	W =  90.000 deg,	P =   0.000 deg,	R =   90.000 deg
};
P[682]{
   GP1:
	UF : 0, UT : 6,		CONFIG : 'N U T, 0, 0, 0',
	X =  232.874  mm,	Y =   -240.688  mm,	Z =   -325.206  mm,
	W =  90.000 deg,	P =   0.000 deg,	R =   90.000 deg
};
P[683]{
   GP1:
	UF : 0, UT : 6,		CONFIG : 'N U T, 0, 0, 0',
	X =  234.528  mm,	Y =   -239.591  mm,	Z =   -311.852  mm,
	W =  90.000 deg,	P =   0.000 deg,	R =   90.000 deg
};
P[684]{
   GP1:
	UF : 0, UT : 6,		CONFIG : 'N U T, 0, 0, 0',
	X =  235.758  mm,	Y =   -238.951  mm,	Z =   -319.159  mm,
	W =  90.000 deg,	P =   0.000 deg,	R =   90.000 deg
};
P[685]{
   GP1:
	UF : 0, UT : 6,		CONFIG : 'N U T, 0, 0, 0',
	X =  236.653  mm,	Y =   -238.797  mm,	Z =   -309.774  mm,
	W =  90.000 deg,	P =   0.000 deg,	R =   90.000 deg
};
P[686]{
   GP1:
	UF : 0, UT : 6,		CONFIG : 'N U T, 0, 0, 0',
	X =  237.094  mm,	Y =   -237.974  mm,	Z =   -322.491  mm,
	W =  90.000 deg,	P =   0.000 deg,	R =   90.000 deg
};
P[687]{
   GP1:
	UF : 0, UT : 6,		CONFIG : 'N U T, 0, 0, 0',
	X =  237.986  mm,	Y =   -237.364  mm,	Z =   -324.620  mm,
	W =  90.000 deg,	P =   0.000 deg,	R =   90.000 deg
};
P[688]{
   GP1:
	UF : 0, UT : 6,		CONFIG : 'N U T, 0, 0, 0',
	X =  238.909  mm,	Y =   -237.029  mm,	Z =   -320.644  mm,
	W =  90.000 deg,	P =   0.000 deg,	R =   90.000 deg
};
P[689]{
   GP1:
	UF : 0, UT : 6,		CONFIG : 'N U T, 0, 0, 0',
	X =  239.607  mm,	Y =   -236.195  mm,	Z =   -318.680  mm,
	W =  90.000 deg,	P =   0.000 deg,	R =   90.000 deg
};
P[690]{
   GP1:
	UF : 0, UT : 6,		CONFIG : 'N U T, 0, 0, 0',
	X =  240.635  mm,	Y =   -236.195  mm,	Z =   -327.317  mm,
	W =  90.000 deg,	P =   0.000 deg,	R =   90.000 deg
};
P[691]{
   GP1:
	UF : 0, UT : 6,		CONFIG : 'N U T, 0, 0, 0',
	X =  241.360  mm,	Y =   -235.612  mm,	Z =   -323.227  mm,
	W =  90.000 deg,	P =   0.000 deg,	R =   90.000 deg
};
P[692]{
   GP1:
	UF : 0, UT : 6,		CONFIG : 'N U T, 0, 0, 0',
	X =  242.700  mm,	Y =   -235.350  mm,	Z =   -313.481  mm,
	W =  90.000 deg,	P =   0.000 deg,	R =   90.000 deg
};
P[693]{
   GP1:
	UF : 0, UT : 6,		CONFIG : 'N U T, 0, 0, 0',
	X =  243.340  mm,	Y =   -234.579  mm,	Z =   -317.524  mm,
	W =  90.000 deg,	P =   0.000 deg,	R =   90.000 deg
};
P[694]{
   GP1:
	UF : 0, UT : 6,		CONFIG : 'N U T, 0, 0, 0',
	X =  243.875  mm,	Y =   -233.814  mm,	Z =   -322.860  mm,
	W =  90.000 deg,	P =   0.000 deg,	R =   90.000 deg
};
P[695]{
   GP1:
	UF : 0, UT : 6,		CONFIG : 'N U T, 0, 0, 0',
	X =  251.685  mm,	Y =   -247.320  mm,	Z =   -319.828  mm,
	W =  90.000 deg,	P =   0.000 deg,	R =   90.000 deg
};
P[696]{
   GP1:
	UF : 0, UT : 6,		CONFIG : 'N U T, 0, 0, 0',
	X =  250.950  mm,	Y =   -247.417  mm,	Z =   -323.833  mm,
	W =  90.000 deg,	P =   0.000 deg,	R =   90.000 deg
};
P[697]{
   GP1:
	UF : 0, UT : 6,		CONFIG : 'N U T, 0, 0, 0',
	X =  249.941  mm,	Y =   -247.905  mm,	Z =   -315.874  mm,
	W =  90.000 deg,	P =   0.000 deg,	R =   90.000 deg
};
P[698]{
   GP1:
	UF : 0, UT : 6,		CONFIG : 'N U T, 0, 0, 0',
	X =  249.286  mm,	Y =   -248.681  mm,	Z =   -326.489  mm,
	W =  90.000 deg,	P =   0.000 deg,	R =   90.000 deg
};
P[699]{
   GP1:
	UF : 0, UT : 6,		CONFIG : 'N U T, 0, 0, 0',
	X =  248.184  mm,	Y =   -249.046  mm,	Z =   -319.997  mm,
	W =  90.000 deg,	P =   0.000 deg,	R =   90.000 deg
};
P[700]{
   GP1:
	UF : 0, UT : 6,		CONFIG : 'N U T, 0, 0, 0',
	X =  247.169  mm,	Y =   -249.764  mm,	Z =   -312.118  mm,
	W =  90.000 deg,	P =   0.000 deg,	R =   90.000 deg
};
P[701]{
   GP1:
	UF : 0, UT : 6,		CONFIG : 'N U T, 0, 0, 0',
	X =  245.857  mm,	Y =   -250.280  mm,	Z =   -320.017  mm,
	W =  90.000 deg,	P =   0.000 deg,	R =   90.000 deg
};
P[702]{
   GP1:
	UF : 0, UT : 6,		CONFIG : 'N U T, 0, 0, 0',
	X =  244.538  mm,	Y =   -250.848  mm,	Z =   -320.296  mm,
	W =  90.000 deg,	P =   0.000 deg,	R =   90.000 deg
};
P[703]{
   GP1:
	UF : 0, UT : 6,		CONFIG : 'N U T, 0, 0, 0',
	X =  243.238  mm,	Y =   -252.075  mm,	Z =   -320.057  mm,
	W =  90.000 deg,	P =   0.000 deg,	R =   90.000 deg
};
P[704]{
   GP1:
	UF : 0, UT : 6,		CONFIG : 'N U T, 0, 0, 0',
	X =  242.208  mm,	Y =   -252.169  mm,	Z =   -315.734  mm,
	W =  90.000 deg,	P =   0.000 deg,	R =   90.000 deg
};
P[705]{
   GP1:
	UF : 0, UT : 6,		CONFIG : 'N U T, 0, 0, 0',
	X =  241.629  mm,	Y =   -253.196  mm,	Z =   -310.770  mm,
	W =  90.000 deg,	P =   0.000 deg,	R =   90.000 deg
};
P[706]{
   GP1:
	UF : 0, UT : 6,		CONFIG : 'N U T, 0, 0, 0',
	X =  240.445  mm,	Y =   -253.552  mm,	Z =   -327.369  mm,
	W =  90.000 deg,	P =   0.000 deg,	R =   90.000 deg
};
P[707]{
   GP1:
	UF : 0, UT : 6,		CONFIG : 'N U T, 0, 0, 0',
	X =  239.253  mm,	Y =   -253.723  mm,	Z =   -312.040  mm,
	W =  90.000 deg,	P =   0.000 deg,	R =   90.000 deg
};
P[708]{
   GP1:
	UF : 0, UT : 6,		CONFIG : 'N U T, 0, 0, 0',
	X =  238.483  mm,	Y =   -254.793  mm,	Z =   -316.964  mm,
	W =  90.000 deg,	P =   0.000 deg,	R =   90.000 deg
};
P[709]{
   GP1:
	UF : 0, UT : 6,		CONFIG : 'N U T, 0, 0, 0',
	X =  237.911  mm,	Y =   -255.445  mm,	Z =   -323.514  mm,
	W =  90.000 deg,	P =   0.000 deg,	R =   90.000 deg
};
P[710]{
   GP1:
	UF : 0, UT : 6,		CONFIG : 'N U T, 0, 0, 0',
	X =  237.275  mm,	Y =   -255.882  mm,	Z =   -317.928  mm,
	W =  90.000 deg,	P =   0.000 deg,	R =   90.000 deg
};
P[711]{
   GP1:
	UF : 0, UT : 6,		CONFIG : 'N U T, 0, 0, 0',
	X =  236.103  mm,	Y =   -256.109  mm,	Z =   -316.019  mm,
	W =  90.000 deg,	P =   0.000 deg,	R =   90.000 deg
};
P[712]{
   GP1:
	UF : 0, UT : 6,		CONFIG : 'N U T, 0, 0, 0',
	X =  234.802  mm,	Y =   -256.309  mm,	Z =   -317.470  mm,
	W =  90.000 deg,	P =   0.000 deg,	R =   90.000 deg
};
P[713]{
   GP1:
	UF : 0, UT : 6,		CONFIG : 'N U T, 0, 0, 0',
	X =  234.479  mm,	Y =   -257.087  mm,	Z =   -310.012  mm,
	W =  90.000 deg,	P =   0.000 deg,	R =   90.000 deg
};
P[714]{
   GP1:
	UF : 0, UT : 6,		CONFIG : 'N U T, 0, 0, 0',
	X =  233.248  mm,	Y =   -257.646  mm,	Z =   -325.932  mm,
	W =  90.000 deg,	P =   0.000 deg,	R =   90.000 deg
};
P[715]{
   GP1:
	UF : 0, UT : 6,		CONFIG : 'N U T, 0, 0, 0',
	X =  232.304  mm,	Y =   -258.623  mm,	Z =   -316.381  mm,
	W =  90.000 deg,	P =   0.000 deg,	R =   90.000 deg
};
P[716]{
   GP1:
	UF : 0, UT : 6,		CONFIG : 'N U T, 0, 0, 0',
	X =  231.494  mm,	Y =   -258.312  mm,	Z =   -318.827  mm,
	W =  90.000 deg,	P =   0.000 deg,	R =   90.000 deg
};
P[717]{
   GP1:
	UF : 0, UT : 6,		CONFIG : 'N U T, 0, 0, 0',
	X =  230.858  mm,	Y =   -258.701  mm,	Z =   -320.224  mm,
	W =  90.000 deg,	P =   0.000 deg,	R =   90.000 deg
};
P[718]{
   GP1:
	UF : 0, UT : 6,		CONFIG : 'N U T, 0, 0, 0',
	X =  230.079  mm,	Y =   -259.361  mm,	Z =   -313.222  mm,
	W =  90.000 deg,	P =   0.000 deg,	R =   90.000 deg
};
P[719]{
   GP1:
	UF : 0, UT : 6,		CONFIG : 'N U T, 0, 0, 0',
	X =  228.888  mm,	Y =   -260.467  mm,	Z =   -324.129  mm,
	W =  90.000 deg,	P =   0.000 deg,	R =   90.000 deg
};
P[720]{
   GP1:
	UF : 0, UT : 6,		CONFIG : 'N U T, 0, 0, 0',
	X =  228.074  mm,	Y =   -260.125  mm,	Z =   -316.510  mm,
	W =  90.000 deg,	P =   0.000 deg,	R =   90.000 deg
};
P[721]{
   GP1:
	UF : 0, UT : 6,		CONFIG : 'N U T, 0, 0, 0',
	X =  227.383  mm,	Y =   -261.268  mm,	Z =   -321.728  mm,
	W =  90.000 deg,	P =   0.000 deg,	R =   90.000 deg
};
P[722]{
   GP1:
	UF : 0, UT : 6,		CONFIG : 'N U T, 0, 0, 0',
	X =  225.660  mm,	Y =   -262.329  mm,	Z =   -326.469  mm,
	W =  90.000 deg,	P =   0.000 deg,	R =   90.000 deg
};
P[723]{
   GP1:
	UF : 0, UT : 6,		CONFIG : 'N U T, 0, 0, 0',
	X =  224.581  mm,	Y =   -263.203  mm,	Z =   -317.101  mm,
	W =  90.000 deg,	P =   0.000 deg,	R =   90.000 deg
};
P[724]{
   GP1:
	UF : 0, UT : 6,		CONFIG : 'N U T, 0, 0, 0',
	X =  223.753  mm,	Y =   -263.618  mm,	Z =   -310.255  mm,
	W =  90.000 deg,	P =   0.000 deg,	R =   90.000 deg
};
P[725]{
   GP1:
	UF : 0, UT : 6,		CONFIG : 'N U T, 0, 0, 0',
	X =  222.500  mm,	Y =   -263.291  mm,	Z =   -316.275  mm,
	W =  90.000 deg,	P =   0.000 deg,	R =   90.000 deg
};
P[726]{
   GP1:
	UF : 0, UT : 6,		CONFIG : 'N U T, 0, 0, 0',
	X =  222.140  mm,	Y =   -263.879  mm,	Z =   -309.986  mm,
	W =  90.000 deg,	P =   0.000 deg,	R =   90.000 deg
};
P[727]{
   GP1:
	UF : 0, UT : 6,		CONFIG : 'N U T, 0, 0, 0',
	X =  221.958  mm,	Y =   -263.600  mm,	Z =   -323.080  mm,
	W =  90.000 deg,	P =   0.000 deg,	R =   90.000 deg
};
P[728]{
   GP1:
	UF : 0, UT : 6,		CONFIG : 'N U T, 0, 0, 0',
	X =  222.206  mm,	Y =   -264.111  mm,	Z =   -309.829  mm,
	W =  90.000 deg,	P =   0.000 deg,	R =   90.000 deg
};
P[729]{
   GP1:
	UF : 0, UT : 6,		CONFIG : 'N U T, 0, 0, 0',
	X =  222.000  mm,	Y =   -263.966  mm,	Z =   -318.016  mm,
	W =  90.000 deg,	P =   0.000 deg,	R =   90.000 deg
};
P[730]{
   GP1:
	UF : 0, UT : 6,		CONFIG : 'N U T, 0, 0, 0',
	X =  221.561  mm,	Y =   -264.742  mm,	Z =   -325.092  mm,
	W =  90.000 deg,	P =   0.000 deg,	R =   90.000 deg
};
P[731]{
   GP1:
	UF : 0, UT : 6,		CONFIG : 'N U T, 0, 0, 0',
	X =  221.313  mm,	Y =   -264.723  mm,	Z =   -323.427  mm,
	W =  90.000 deg,	P =   0.000 deg,	R =   90.000 deg
};
P[732]{
   GP1:
	UF : 0, UT : 6,		CONFIG : 'N U T, 0, 0, 0',
	X =  221.205  mm,	Y =   -264.556  mm,	Z =   -321.557  mm,
	W =  90.000 deg,	P =   0.000 deg,	R =   90.000 deg
};
P[733]{
   GP1:
	UF : 0, UT : 6,		CONFIG : 'N U T, 0, 0, 0',
	X =  221.306  mm,	Y =   -265.009  mm,	Z =   -318.376  mm,
